// TwinCAT 3 PLC project Fraktal_Tests
// Title: Fraktal_Tests
// Company: fraktal-automation
// Author: fraktal-automation
// ProjectVersion: 0.1.0.10
// Description: Aggregate Fraktal Core + Modules + Press Demo TcUnit gate - excluded from deployed runtime (Core 5.7).
// ProgramVersion: 3.1.4026.24
// libraries:
//   Tc2_Standard, * (Beckhoff Automation GmbH)
//   Tc2_System, * (Beckhoff Automation GmbH)
//   Tc2_Utilities, * (Beckhoff Automation GmbH)
//   Tc3_Module, * (Beckhoff Automation GmbH)
//   Fraktal_Core, 0.3.0.0 (fraktal-automation)
//   Fraktal_Modules, 0.2.0.0 (fraktal-automation)
//   TcUnit, * (www.tcunit.org)
// project tree:
//   / PlcTask.TcTTO (not stored), FB_Access_Tests.TcPOU (not stored), FB_AlarmLog_Tests.TcPOU (not stored), FB_Base_Tests.TcPOU (not stored), FB_FaultRecovery_Tests.TcPOU, FB_ConfigurableCylinderCM_Tests.TcPOU (not stored), FB_ClampEM_Tests.TcPOU, FB_ClampStationUnit_Tests.TcPOU (not stored), FB_Connector_Tests.TcPOU (not stored), FB_CylinderCM_Tests.TcPOU, FB_Decision_Tests.TcPOU, FB_Hmi_Tests.TcPOU, FB_IoTopologyPublisher_Tests.TcPOU (not stored), FB_InputCM_Tests.TcPOU (not stored), FB_ManualCmd_Tests.TcPOU (not stored), FB_MultiRoot_Tests.TcPOU (not stored), FB_Oee_Tests.TcPOU (not stored), FB_PermIntlk_Tests.TcPOU (not stored), FB_PowerGroupCM_Tests.TcPOU (not stored), FB_TwoHandStartCM_Tests.TcPOU (not stored), FB_PressDemoUnit_Tests.TcPOU (not stored), FB_ProbeCM.TcPOU (not stored), FB_ProbeConnector.TcPOU (not stored), FB_ProbeEM.TcPOU (not stored), FB_ProbeUnit.TcPOU, FB_ProbeUnitManual.TcPOU (not stored), FB_Release_Tests.TcPOU (not stored), FB_PartTrace_Tests.TcPOU (not stored), FB_Shelve_Tests.TcPOU (not stored), FB_SystemInfrastructure_Tests.TcPOU (not stored), FB_TcpDev_Tests.TcPOU, FB_Timing_Tests.TcPOU (not stored), FB_Unit_Tests.TcPOU, PRG_TcUnitRunner.TcPOU
//   ../Fraktal_Press_Demo/01_PneumaticPress/Sequences/ FB_PressDemoLoadPosition.TcPOU (not stored), FB_PressDemoHome.TcPOU (not stored), FB_PressDemoChangeover.TcPOU (not stored), FB_PressDemoAuto.TcPOU
//   ../Fraktal_Press_Demo/01_PneumaticPress/Release/ FB_PressDemoRelease.TcPOU (not stored)
//   ../Fraktal_Press_Demo/01_PneumaticPress/ FB_PressDemoUnit.TcPOU
// (motion and I/O tree: see PLC project fraktal_press_demo)
// real-time tasks:
//   TASK PlcTask: cycle T#10ms, priority 20, ADS port 350
// variable links:

// ---- ../Fraktal_Press_Demo/01_PneumaticPress/Sequences/FB_PressDemoAuto.TcPOU
// AUTO mode chain (Core §6.2/§6.8 ST skeleton on FB_SequenceBase): the continuous
// production cycle — await a fresh two-hand start with part+air present, transfer
// the part in, press for the recipe dwell, return to load position, count the good
// part, and loop until Stop. A Stop requested at the between-cycles wait is honored
// there (M_StopNow) so no phantom cycle is charged. Every child motion goes through
// the §6.1 handshake (M_MayIssue); progression rides the shared _retVal.
FUNCTION_BLOCK FB_PressDemoAuto EXTENDS FB_SequenceBase
VAR
    _partReady, _airReady, _startReady : BOOL;
    _dwellTwoHandHeld : BOOL;          // N220 named wait: two-hand held through the dwell
    _traceAccepted, _recordAccepted, _partProcessed : BOOL;
    {attribute 'OPC.UA.DA' := '0'}
    _pressRam : REFERENCE TO FB_CylinderCM;
    {attribute 'OPC.UA.DA' := '0'}
    _door : REFERENCE TO FB_CylinderCM;
    {attribute 'OPC.UA.DA' := '0'}
    _partSlide : REFERENCE TO FB_CylinderCM;
    {attribute 'OPC.UA.DA' := '0'}
    _twoHand : REFERENCE TO FB_TwoHandStartCM;
    {attribute 'OPC.UA.DA' := '0'}
    _partPresentSensor : REFERENCE TO FB_DigitalInputCM;
    {attribute 'OPC.UA.DA' := '0'}
    _airPressureMonitor : REFERENCE TO FB_AirPressureMonitorCM;
    {attribute 'OPC.UA.DA' := '0'}
    _parCfg : REFERENCE TO ST_PneumaticPressParCfg;
    {attribute 'OPC.UA.DA' := '0'}
    _outCmd : REFERENCE TO ST_PneumaticPressOutCmd;
    {attribute 'OPC.UA.DA' := '0'}
    _startLatched : REFERENCE TO BOOL;
    {attribute 'OPC.UA.DA' := '0'}
    _loadPosition : FB_PressDemoLoadPosition;
    _loadPositionRunning : BOOL;
END_VAR

METHOD M_Reset
M_ResetBase(0);
_loadPositionRunning := FALSE;
_loadPosition.M_Reset(BaseStepNo := 0);
END_METHOD

METHOD M_Run
IF NOT _attached THEN
    RETURN;
END_IF
CASE _step OF
    0:  // initialize
        M_Step(StepNo := 0, StepName := 'project.step.pressAutoInitialize',
            Awaits := 0, AwaitingLabel := '', TimeClass := E_TimeClass.WORK, ExpectedTime := T#0S);
        _outCmd.CycleCompleted := FALSE;
        _outCmd.Homed := FALSE;
        _outCmd.ChangeoverCompleted := FALSE;
        _loadPositionRunning := FALSE;
        _retVal := E_StepResult.ADVANCE;
        M_Advance(OnAdvance := 100, OnJump1 := -1, OnJump2 := -1, OnJump3 := -1);
    100:  // await a fresh two-hand start (the §8.11.1 cycle-start marker)
        M_Step(StepNo := 100, StepName := 'project.step.pressAwaitTwoHand',
            Awaits := 0, AwaitingLabel := '', TimeClass := E_TimeClass.WAIT_OPERATOR, ExpectedTime := T#0S);
        _outCmd.CycleCompleted := FALSE;
        _partReady := M_Await(Idx := 1, Label := 'project.condition.partPresent',
            Ok := _partPresentSensor.OutImm.Value AND _partPresentSensor.OutImm.Quality);
        _airReady := M_Await(Idx := 2, Label := 'project.condition.airPressureOk',
            Ok := _airPressureMonitor.OutImm.PressureOk);
        IF _parCfg.RequireTwoHandStart THEN
            _startReady := M_Await(Idx := 3, Label := 'project.condition.twoHandStart', Ok := _startLatched);
        ELSE
            _startReady := TRUE;
        END_IF
        IF M_StopPending() THEN
            M_StopNow();                       // stop accepted BETWEEN cycles: no phantom cycle
        ELSIF _partReady AND _airReady AND _startReady THEN
            _traceAccepted := M_PartReceived();
            _retVal := E_StepResult.ADVANCE;
        END_IF
        M_Advance(OnAdvance := 110, OnJump1 := -1, OnJump2 := -1, OnJump3 := -1);
    110:  // ram up
        M_Step(StepNo := 110, StepName := 'project.step.pressRamUp',
            Awaits := _pressRam, AwaitingLabel := 'PressRam.RETRACT', TimeClass := E_TimeClass.WORK, ExpectedTime := T#0S);
        IF M_MayIssue(Steppable := TRUE) THEN
            _pressRam.Abort := FALSE; _pressRam.Command := E_CylinderCommand.RETRACT; _pressRam.Execute := TRUE;
        END_IF
        IF _pressRam.Done THEN _pressRam.Execute := FALSE; _retVal := E_StepResult.ADVANCE; END_IF
        M_Advance(OnAdvance := 130, OnJump1 := -1, OnJump2 := -1, OnJump3 := -1);
    130:  // door open
        M_Step(StepNo := 130, StepName := 'project.step.pressDoorOpen',
            Awaits := _door, AwaitingLabel := 'Door.RETRACT', TimeClass := E_TimeClass.WORK, ExpectedTime := T#0S);
        IF M_MayIssue(Steppable := TRUE) THEN
            _door.Abort := FALSE; _door.Command := E_CylinderCommand.RETRACT; _door.Execute := TRUE;
        END_IF
        IF _door.Done THEN _door.Execute := FALSE; _retVal := E_StepResult.ADVANCE; END_IF
        M_Advance(OnAdvance := 150, OnJump1 := -1, OnJump2 := -1, OnJump3 := -1);
    150:  // slide inside (value-adding sequence begins)
        M_Step(StepNo := 150, StepName := 'project.step.pressSlideInside',
            Awaits := _partSlide, AwaitingLabel := 'PartSlide.EXTEND', TimeClass := E_TimeClass.WORK, ExpectedTime := T#0S);
        IF M_MayIssue(Steppable := TRUE) THEN
            M_PartStarted();
            _partSlide.Abort := FALSE; _partSlide.Command := E_CylinderCommand.EXTEND; _partSlide.Execute := TRUE;
        END_IF
        IF _partSlide.Done THEN _partSlide.Execute := FALSE; _retVal := E_StepResult.ADVANCE; END_IF
        M_Advance(OnAdvance := 170, OnJump1 := -1, OnJump2 := -1, OnJump3 := -1);
    170:  // transfer settle
        M_Step(StepNo := 170, StepName := 'project.step.pressTransferSettle',
            Awaits := 0, AwaitingLabel := '', TimeClass := E_TimeClass.WORK, ExpectedTime := _parCfg.TransferSettleTime);
        _retVal := M_Delay(PT := _parCfg.TransferSettleTime);
        M_Advance(OnAdvance := 180, OnJump1 := -1, OnJump2 := -1, OnJump3 := -1);
    180:  // door close
        M_Step(StepNo := 180, StepName := 'project.step.pressDoorClose',
            Awaits := _door, AwaitingLabel := 'Door.EXTEND', TimeClass := E_TimeClass.WORK, ExpectedTime := T#0S);
        IF M_MayIssue(Steppable := TRUE) THEN
            _door.Abort := FALSE; _door.Command := E_CylinderCommand.EXTEND; _door.Execute := TRUE;
        END_IF
        IF _door.Done THEN _door.Execute := FALSE; _retVal := E_StepResult.ADVANCE; END_IF
        M_Advance(OnAdvance := 200, OnJump1 := -1, OnJump2 := -1, OnJump3 := -1);
    200:  // ram down
        M_Step(StepNo := 200, StepName := 'project.step.pressRamDown',
            Awaits := _pressRam, AwaitingLabel := 'PressRam.EXTEND', TimeClass := E_TimeClass.WORK, ExpectedTime := T#0S);
        IF M_MayIssue(Steppable := TRUE) THEN
            _pressRam.Abort := FALSE; _pressRam.Command := E_CylinderCommand.EXTEND; _pressRam.Execute := TRUE;
        END_IF
        IF _pressRam.Done THEN _pressRam.Execute := FALSE; _retVal := E_StepResult.ADVANCE; END_IF
        M_Advance(OnAdvance := 220, OnJump1 := -1, OnJump2 := -1, OnJump3 := -1);
    220:  // press dwell — two-hand must stay held; releasing it HOLDS the dwell
        M_Step(StepNo := 220, StepName := 'project.step.pressDwell',
            Awaits := 0, AwaitingLabel := '', TimeClass := E_TimeClass.WORK, ExpectedTime := _parCfg.PressSettleTime);
        // Releasing the button mid-dwell is the designed way to stop pressing, so it
        // is a named wait (§6.9(b)), not a fault: the ram's outputs come off, the
        // dwell timer freezes where it is because M_Delay is not called, and pressing
        // again restores the force and finishes the remaining dwell. Faulting here
        // charged an unrecoverable downtime event for normal operator behaviour.
        _dwellTwoHandHeld := M_Await(Idx := 1, Label := 'project.condition.twoHandHeldDuringPress',
            Ok := _twoHand.OutImm.SafeActive OR NOT _parCfg.RequireTwoHandStart);
        IF NOT _dwellTwoHandHeld THEN
            _pressRam.WithdrawOutputs();
        ELSE
            // The press force is the valve latched by the EXTEND that step 200 already
            // completed, so after a withdraw only this call re-energizes it — and the
            // ram re-checks its own extend permit before it does (§7.2).
            _pressRam.RestoreOutputs();
            _retVal := M_Delay(PT := _parCfg.PressSettleTime);
        END_IF
        M_Advance(OnAdvance := 230, OnJump1 := -1, OnJump2 := -1, OnJump3 := -1);
    230:  // record the applied dwell (§3.16.1 measured value)
        M_Step(StepNo := 230, StepName := 'project.step.pressRecordResult',
            Awaits := 0, AwaitingLabel := '', TimeClass := E_TimeClass.WORK, ExpectedTime := T#0S);
        _recordAccepted := M_PartRecord(RecordName := 'PressDwell',
            Value := DINT_TO_LREAL(TIME_TO_DINT(_parCfg.PressSettleTime)),
            Minimum := 0, Maximum := 30000,
            Target := DINT_TO_LREAL(TIME_TO_DINT(_parCfg.PressSettleTime)), EngUnit := 'ms');
        _loadPositionRunning := FALSE;
        _retVal := E_StepResult.ADVANCE;
        M_Advance(OnAdvance := 240, OnJump1 := -1, OnJump2 := -1, OnJump3 := -1);
    240:  // return to the shared load-safe position (composite step)
        IF NOT _loadPositionRunning THEN
            _loadPosition.M_Reset(BaseStepNo := 240);
            _loadPositionRunning := TRUE;
        END_IF
        _loadPosition.M_Run();
        IF _loadPosition.Done THEN
            _loadPositionRunning := FALSE;
            _retVal := E_StepResult.ADVANCE;
        END_IF
        M_Advance(OnAdvance := 999, OnJump1 := -1, OnJump2 := -1, OnJump3 := -1);
    999:  // cycle complete — write result, count by verdict, loop (§8.11.1 finish marker)
        M_Step(StepNo := 999, StepName := 'project.step.pressAutoComplete',
            Awaits := 0, AwaitingLabel := '', TimeClass := E_TimeClass.WORK, ExpectedTime := T#0S);
        _outCmd.CycleCompleted := TRUE;
        _partProcessed := M_PartProcessed(Verdict := E_Verdict.OK, Reason := E_Reason.NONE);
        IF NOT _partProcessed THEN
            M_CountGood();                     // §3.9: no carrier configured — count directly
        END_IF
        _startLatched := FALSE;
        IF M_EndOfCycle() THEN
            _retVal := E_StepResult.ADVANCE;   // stop NOT requested: loop to N100
        END_IF
        M_Advance(OnAdvance := 100, OnJump1 := -1, OnJump2 := -1, OnJump3 := -1);
ELSE
    M_Fault(Reason := E_Reason.STEP_STALLED, DescriptionKey := 'std.error.undefinedStep');
END_CASE
END_METHOD

METHOD Setup : BOOL
VAR_INPUT
    Host : I_SequenceHost;
END_VAR
VAR_IN_OUT
    PressRam : FB_CylinderCM;
    Door : FB_CylinderCM;
    PartSlide : FB_CylinderCM;
    TwoHand : FB_TwoHandStartCM;
    PartPresentSensor : FB_DigitalInputCM;
    AirPressureMonitor : FB_AirPressureMonitorCM;
    ParCfg : ST_PneumaticPressParCfg;
    OutCmd : ST_PneumaticPressOutCmd;
    StartLatched : BOOL;
END_VAR
_pressRam REF= PressRam;
_door REF= Door;
_partSlide REF= PartSlide;
_twoHand REF= TwoHand;
_partPresentSensor REF= PartPresentSensor;
_airPressureMonitor REF= AirPressureMonitor;
_parCfg REF= ParCfg;
_outCmd REF= OutCmd;
_startLatched REF= StartLatched;
Setup := M_Attach(Host := Host) AND __ISVALIDREF(_pressRam) AND __ISVALIDREF(_door)
    AND __ISVALIDREF(_partSlide) AND __ISVALIDREF(_twoHand)
    AND __ISVALIDREF(_partPresentSensor) AND __ISVALIDREF(_airPressureMonitor)
    AND __ISVALIDREF(_parCfg) AND __ISVALIDREF(_outCmd) AND __ISVALIDREF(_startLatched)
    AND _loadPosition.Setup(Host := Host, PressRam := PressRam, Door := Door, PartSlide := PartSlide);
END_METHOD

END_FUNCTION_BLOCK

// ---- ../Fraktal_Press_Demo/01_PneumaticPress/FB_PressDemoUnit.TcPOU
// Project-owned Unit: pneumatic press + access door + transfer slide + two-hand request.
// Cylinder interlocks prevent the two documented collisions in AUTO and MANUAL.
// Certified E-stop, two-hand evaluation and safe valve outputs remain external.
FUNCTION_BLOCK FB_PressDemoUnit EXTENDS FB_UnitBase
VAR_INPUT
    ParCfg : ST_PneumaticPressParCfg;
    ParCmd : ST_PneumaticPressParCmd;
END_VAR
VAR_OUTPUT
    PressRam      : FB_CylinderCM;
    Door          : FB_CylinderCM;
    PartSlide     : FB_CylinderCM;
    TwoHand       : FB_TwoHandStartCM;
    PneumaticPower: FB_PowerGroupCM;
    PartPresentSensor : FB_DigitalInputCM;
    AirPressureMonitor : FB_AirPressureMonitorCM;
    ReleaseConditions : FB_PressDemoRelease; // project-owned, browseable condition state
    OutCmd        : ST_PneumaticPressOutCmd;
    OutImm        : ST_PneumaticPressOutImm;
END_VAR
VAR
    {attribute 'OPC.UA.DA' := '0'}
    _recipe : I_RecipeProvider;
    _parCfgStaged : ST_PneumaticPressParCfg;
    _recipePrepared : BOOL;
    _startLatched : BOOL;
    _powerRequestPending : BOOL;
    _powerTargetOn : BOOL;
    {attribute 'OPC.UA.DA' := '0'}
    _homeSequence : FB_PressDemoHome;       // §6.8 ST chain on FB_SequenceBase owns HOME steps
    {attribute 'OPC.UA.DA' := '0'}
    _changeoverSequence : FB_PressDemoChangeover;
    {attribute 'OPC.UA.DA' := '0'}
    _autoSequence : FB_PressDemoAuto;
END_VAR

Cyclic();

METHOD Setup : BOOL
VAR_INPUT
    Name : STRING(80);
    PressHal : REFERENCE TO ST_CylinderHal;
    DoorHal : REFERENCE TO ST_CylinderHal;
    SlideHal : REFERENCE TO ST_CylinderHal;
    TwoHandHal : REFERENCE TO ST_TwoHandHal;
    PowerHal : REFERENCE TO ST_PowerGroupHal;
    PartPresentHal : REFERENCE TO ST_DigitalInputHal;
    AirPressureHal : REFERENCE TO ST_AirPressureHal;
    Recipe : I_RecipeProvider;
END_VAR
VAR
    InitialModel : ST_ModelId;
    Ok : BOOL;
END_VAR
_M_SetName(Name);
_M_SetPresentation(DisplayNameKey := 'project.module.pneumaticPress.name', DescriptionKey := 'project.module.pneumaticPress.description');
_recipe := Recipe;
Ok := PressRam.Setup(Name := CONCAT(Name, '.PressRam'), HalRef := PressHal, Recipe := 0);
Ok := Door.Setup(Name := CONCAT(Name, '.Door'), HalRef := DoorHal, Recipe := 0) AND Ok;
Ok := PartSlide.Setup(Name := CONCAT(Name, '.PartSlide'), HalRef := SlideHal, Recipe := 0) AND Ok;
Ok := TwoHand.Setup(Name := CONCAT(Name, '.TwoHand'), HalRef := TwoHandHal) AND Ok;
Ok := PneumaticPower.Setup(Name := CONCAT(Name, '.PneumaticPower'), HalRef := PowerHal) AND Ok;
Ok := PartPresentSensor.Setup(Name := CONCAT(Name, '.PartPresentSensor'),
    HalRef := PartPresentHal, DisplayNameKey := 'project.module.partPresentSensor.name',
    DescriptionKey := 'project.module.partPresentSensor.description') AND Ok;
Ok := AirPressureMonitor.Setup(Name := CONCAT(Name, '.AirPressureMonitor'),
    HalRef := AirPressureHal) AND Ok;
Ok := ReleaseConditions.Setup(UnitPath := Name) AND Ok;
Ok := _homeSequence.Setup(Host := THIS^, PressRam := PressRam, Door := Door,
    PartSlide := PartSlide, OutCmd := OutCmd) AND Ok;
Ok := _changeoverSequence.Setup(Host := THIS^, PressRam := PressRam, Door := Door,
    PartSlide := PartSlide, OutCmd := OutCmd, Model := Model) AND Ok;
Ok := _autoSequence.Setup(Host := THIS^, PressRam := PressRam, Door := Door,
    PartSlide := PartSlide, TwoHand := TwoHand, PartPresentSensor := PartPresentSensor,
    AirPressureMonitor := AirPressureMonitor, ParCfg := ParCfg, OutCmd := OutCmd,
    StartLatched := _startLatched) AND Ok;
PneumaticPower.ParCfg.Kind := E_PowerGroupKind.VALVE_ZONE;
PneumaticPower.ParCfg.RequiredForControl := TRUE;
PneumaticPower.ParCfg.FieldbusLossReaction := E_FieldbusLossReaction.CONTROL_OFF;
Ok := _M_Register(PressRam) AND Ok;
Ok := _M_Register(Door) AND Ok;
Ok := _M_Register(PartSlide) AND Ok;
Ok := _M_Register(TwoHand) AND Ok;
Ok := _M_Register(PneumaticPower) AND Ok;
Ok := _M_Register(PartPresentSensor) AND Ok;
Ok := _M_Register(AirPressureMonitor) AND Ok;
Setup := Ok AND PrepareRecipe(Model := InitialModel);
IF Setup THEN CommitRecipe(); END_IF
END_METHOD

METHOD PrepareRecipe : BOOL
VAR_INPUT
    Model : ST_ModelId;
END_VAR
IF _recipe = 0 THEN
    _parCfgStaged := ParCfg;
    _recipePrepared := TRUE;
ELSIF _recipe.Load(ModelCode := Model.ModelCode, RecipeKey := 'PneumaticPressUnit', pParCfg := ADR(_parCfgStaged), Size := SIZEOF(_parCfgStaged)) THEN
    IF (_parCfgStaged.PressSettleTime > T#30S) OR (_parCfgStaged.TransferSettleTime > T#5S) THEN
        _M_Fault(E_Reason.RECIPE_INVALID, 'project.error.pressRecipeInvalid');
        _recipePrepared := FALSE;
        PrepareRecipe := FALSE;
        RETURN;
    END_IF
    _recipePrepared := TRUE;
ELSE
    _M_Fault(E_Reason.RECIPE_INVALID, 'std.error.recipeSchemaInvalid');
    _recipePrepared := FALSE;
    PrepareRecipe := FALSE;
    RETURN;
END_IF
PrepareRecipe := SUPER^.PrepareRecipe(Model := Model);
IF NOT PrepareRecipe THEN _recipePrepared := FALSE; END_IF
END_METHOD

METHOD CommitRecipe
SUPER^.CommitRecipe();
IF _recipePrepared THEN
    ParCfg := _parCfgStaged;
    // §8.11 performance references follow the model: OEE Performance denominator
    // and the WORK-time degradation baseline are per-recipe engineering data.
    Oee.IdealCycleMs := ParCfg.IdealCycleMs;
    Profiler.M_SetBaselineWork(WorkMs := ParCfg.BaselineWorkMs);
END_IF
_recipePrepared := FALSE;
END_METHOD

METHOD AbortRecipe
SUPER^.AbortRecipe();
_recipePrepared := FALSE;
END_METHOD

// First operational scan: initialize application-owned mode-chain state.
METHOD PROTECTED OnInit : DINT
OnInit := SUPER^.OnInit();
_M_ResetModeSequences();
_M_ClearModeTransitionState();
END_METHOD

// Every accepted Unit Start gets a fresh mode chain, including a repeated
// HOME/CHANGEOVER run that does not pass through another mode change.
METHOD PROTECTED OnCommandStart : DINT
OnCommandStart := SUPER^.OnCommandStart();
_M_ResetModeSequences();
END_METHOD

// Mode-entry wiring only. Step behavior remains in the selected sequence POU.
METHOD PROTECTED OnModeChanged : DINT
VAR_INPUT
    NewMode : E_Mode;
    OldMode : E_Mode;
END_VAR
OnModeChanged := SUPER^.OnModeChanged(
    NewMode := NewMode, OldMode := OldMode);
_M_ResetModeSequences();
_M_ClearModeTransitionState();
END_METHOD

METHOD PROTECTED OnCyclic : DINT
OnCyclic := SUPER^.OnCyclic();
// Project release engineering is a separate visible component. It owns the
// functional collision permits and mode-entry conditions consumed below.
ReleaseConditions.M_Evaluate(PressRam := PressRam, Door := Door, PartSlide := PartSlide,
    TwoHand := TwoHand, PneumaticPower := PneumaticPower,
    AirPressure := AirPressureMonitor);

// Latch access-gated Unit requests, then observe one full Execute-low scan before
// starting another power-group command (PLCopen edge discipline).
IF ControlOffRequest THEN
    _powerTargetOn := FALSE;
    _powerRequestPending := TRUE;
ELSIF ControlOnRequest THEN
    _powerTargetOn := TRUE;
    _powerRequestPending := TRUE;
END_IF
IF PneumaticPower.Done OR PneumaticPower.Error OR PneumaticPower.Aborted THEN
    PneumaticPower.Execute := FALSE;
ELSIF _powerRequestPending AND NOT PneumaticPower.Execute
AND (PneumaticPower.State = E_ExecState.READY) THEN
    PneumaticPower.Abort := FALSE;
    IF _powerTargetOn THEN
        PneumaticPower.Command := E_PowerGroupCommand.POWER_ON;
    ELSE
        PneumaticPower.Command := E_PowerGroupCommand.POWER_OFF;
    END_IF
    PneumaticPower.Execute := TRUE;
    _powerRequestPending := FALSE;
END_IF

// A physical two-hand edge may start AUTO from READY, or release an already
// running Unit's wait step. It never bypasses domain readiness or access policy.
IF TwoHand.OutImm.StartPulse
AND PartPresentSensor.OutImm.Value AND PartPresentSensor.OutImm.Quality
AND AirPressureMonitor.OutImm.PressureOk THEN
    IF (State = E_ExecState.BUSY) AND (ModeActive = E_Mode.AUTO) THEN
        _startLatched := TRUE;
    ELSIF (ModeActive = E_Mode.AUTO) AND Start() THEN
        _startLatched := TRUE;
    END_IF
ELSIF TwoHand.OutImm.StartPulse THEN
    _startLatched := FALSE;
END_IF
IF PneumaticPower.Error AND (State = E_ExecState.BUSY) THEN
    _M_RollupFault();
END_IF
IF (State = E_ExecState.BUSY)
AND NOT AirPressureMonitor.OutImm.PressureOk THEN
    PressRam.WithdrawOutputs();
    Door.WithdrawOutputs();
    PartSlide.WithdrawOutputs();
    _M_Fault(E_Reason.PERMISSIVE_NOT_MET, 'project.error.pressAirPressureLost');
END_IF
OutImm.PressRetracted := PressRam.OutImm.Retracted;
OutImm.DoorOpen := Door.OutImm.Retracted;
OutImm.DoorClosed := Door.OutImm.Extended;
OutImm.SlideInside := PartSlide.OutImm.Extended;
OutImm.SlideOutside := PartSlide.OutImm.Retracted;
OutImm.TwoHandArmed := TwoHand.OutImm.Armed;
OutImm.TwoHandActive := TwoHand.OutImm.SafeActive;
OutImm.PartPresent := PartPresentSensor.OutImm.Value AND PartPresentSensor.OutImm.Quality;
OutImm.AirPressureOk := AirPressureMonitor.OutImm.PressureOk;
OutImm.ReadyForLoad := Door.OutImm.Retracted AND NOT Door.OutImm.Extended
    AND PartSlide.OutImm.Retracted AND NOT PartSlide.OutImm.Extended
    AND PressRam.OutImm.Retracted AND NOT PressRam.OutImm.Extended;
OutImm.ActiveSettleTime := ParCfg.PressSettleTime;
OutImm.Diagnostic := Status.Diagnostic;
END_METHOD

METHOD PROTECTED OnAbort : DINT
OnAbort := SUPER^.OnAbort();
_M_PartAborted();                    // §3.16.3: the part leaves without a valid result
_M_WithdrawSequenceOutputs();
_M_ResetModeSequences();
_M_ClearModeTransitionState();
_powerTargetOn := FALSE;
_powerRequestPending := TRUE;
END_METHOD

// Error-state Abort is a deliberate recovery action but does not clear ERROR.
METHOD PROTECTED OnAbortInError : DINT
OnAbortInError := SUPER^.OnAbortInError();
_M_WithdrawSequenceOutputs();
_M_ResetModeSequences();
_M_ClearModeTransitionState();
_powerTargetOn := FALSE;
_powerRequestPending := TRUE;
END_METHOD

// An operator reset is recovering this Unit: put the application back to the same
// safe wiring an error-state abort establishes, so the reset the operator presses at
// the panel needs no separate Stop/Abort first. The base then releases the run
// command and the children's commands, so the next HOME gets a genuine command edge.
// Unlike the abort paths this does NOT touch control power in either direction: it
// never requests Control On (§9.8 forbids self-resume), and it must not request
// Control Off either — powering down a healthy control circuit would make the
// operator re-enable it before HOME could run, i.e. reintroduce the multi-action
// recovery this reset exists to remove. Power stays where the operator put it.
METHOD PROTECTED OnOperatorReset : DINT
OnOperatorReset := SUPER^.OnOperatorReset();
_M_WithdrawSequenceOutputs();
_M_ResetModeSequences();
_M_ClearModeTransitionState();
END_METHOD

// One safe-stop wiring point shared by normal and error-state abort transitions.
METHOD PROTECTED _M_WithdrawSequenceOutputs
PressRam.WithdrawOutputs();
Door.WithdrawOutputs();
PartSlide.WithdrawOutputs();
PressRam.Execute := FALSE;
Door.Execute := FALSE;
PartSlide.Execute := FALSE;
END_METHOD

// Reset application-owned chain plumbing at lifecycle transitions. The chains'
// N000/N999 steps remain the only owners of process initialization/completion.
METHOD PROTECTED _M_ResetModeSequences
_homeSequence.M_Reset();
_changeoverSequence.M_Reset();
_autoSequence.M_Reset();
END_METHOD

// Clear state that must not survive init, mode entry, or either abort path.
// OnCommandStart deliberately does not call this: a physical start pulse may have
// been latched one scan before the inherited Execute edge is consumed.
METHOD PROTECTED _M_ClearModeTransitionState
Decision.Prompt := '';
DecisionAnswer := 0;
_startLatched := FALSE;
END_METHOD

// Application-only seam for ordinary hardwired Control On/Off buttons.
// It is a method (not OPC UA data), so HMI writes still use the access-gated
// ReqControlOn/ReqControlOff contract. The power CM rechecks safety and health.
METHOD RequestLocalControl : BOOL
VAR_INPUT
    ControlOn : BOOL;
END_VAR
_powerTargetOn := ControlOn;
_powerRequestPending := TRUE;
RequestLocalControl := TRUE;
END_METHOD

// §3.4.2 — the press paces every motion boundary through _M_StepGate, so
// SINGLE_STEP and HOLD_TO_RUN are supported (NON-SAFETY pacing; interlocks
// and the certified safety layer are unaffected).
METHOD PROTECTED _M_SupportsRunStyle : BOOL
VAR_INPUT
    Style : E_RunStyle;
END_VAR
_M_SupportsRunStyle := (Style = E_RunStyle.CONTINUOUS)
    OR (Style = E_RunStyle.SINGLE_STEP) OR (Style = E_RunStyle.HOLD_TO_RUN);
END_METHOD

METHOD PROTECTED _M_Supports : BOOL
VAR_INPUT
    Mode : E_Mode;
END_VAR
_M_Supports := (Mode = E_Mode.AUTO) OR (Mode = E_Mode.MANUAL)
    OR (Mode = E_Mode.HOME) OR (Mode = E_Mode.CHANGEOVER);
END_METHOD

// Thin mode router. Each supported sequence is a named method in the Unit tree.
METHOD PROTECTED _M_Dispatch
CASE ModeActive OF
    E_Mode.AUTO:
        _M_SequenceAuto();
    E_Mode.HOME:
        _M_SequenceHome();
    E_Mode.CHANGEOVER:
        _M_SequenceChangeover();
    E_Mode.MANUAL:
        _M_Fault(E_Reason.UNSUPPORTED_COMMAND, 'project.error.pressManualHasNoSequence');
ELSE
    _M_Fault(E_Reason.UNSUPPORTED_COMMAND, 'project.error.pressModeHasNoSequence');
END_CASE
END_METHOD

// Wiring-only HOME adapter. OnCommandStart owns the reset edge; the sequence POU
// owns every process step and terminal action.
METHOD PROTECTED _M_SequenceHome
_homeSequence.M_Run();
END_METHOD

// Wiring-only CHANGEOVER adapter. The §6.8 chain owns model validation, safe
// positioning, the operator decision, and completion logic.
METHOD PROTECTED _M_SequenceChangeover
_changeoverSequence.M_Run();
END_METHOD

// Wiring-only AUTO adapter. Every production command, wait, timer, decision,
// traceability action, and transition lives in the §6.8 chain.
METHOD PROTECTED _M_SequenceAuto
_autoSequence.M_Run();
END_METHOD

METHOD PROTECTED _M_RouteManual : BOOL
VAR_INPUT
    TargetPath : STRING(255);
    Value : DINT;
END_VAR
_M_RouteManual := FALSE;
IF TargetPath = PressRam.Name THEN
    _M_RouteManual := PressRam.ManualCommand(Value := Value);
ELSIF TargetPath = Door.Name THEN
    _M_RouteManual := Door.ManualCommand(Value := Value);
ELSIF TargetPath = PartSlide.Name THEN
    _M_RouteManual := PartSlide.ManualCommand(Value := Value);
ELSE
    _M_RouteManual := FALSE;
END_IF
END_METHOD

// §7.8 mode-entry release owned by this Unit. The base Start method consumes the
// same report the HMI displays, so this condition cannot become explanation-only.
METHOD PROTECTED _M_AppendInterlocks
VAR_IN_OUT
    Report : ST_ReleaseReport;
END_VAR
ReleaseConditions.M_AppendStart(Report := Report);
END_METHOD

METHOD PROTECTED _M_AppendManualInterlocks
VAR_INPUT
    TargetPath : STRING(255);
    Value : DINT;
END_VAR
VAR_IN_OUT
    Report : ST_ReleaseReport;
END_VAR
ReleaseConditions.M_AppendManual(TargetPath := TargetPath, Value := Value,
    PressRam := PressRam, Door := Door, PartSlide := PartSlide, Report := Report);
END_METHOD

METHOD PROTECTED _M_PublishStatus
SUPER^._M_PublishStatus();
OutImm.Diagnostic := Status.Diagnostic;
END_METHOD

// §3.10.2 — base walk (Unit facets + all child modules), then the project-owned
// fieldbus topology identity: static members of GVL_PressFieldbus.Topology are
// OPC.UA.DA=0 and reach the HMI only through this manifest.
METHOD M_AppendConfig : BOOL
VAR_INPUT
    Pager : REFERENCE TO FB_ConfigPager;
END_VAR
M_AppendConfig := SUPER^.M_AppendConfig(Pager := Pager);
F_AppendTopologyConfig(Topology := GVL_PressFieldbus.Topology, Pager := Pager);
END_METHOD

END_FUNCTION_BLOCK

// ---- FB_FaultRecovery_Tests.TcPOU
// Regression suite for the press hard-lock: an AUTO cycle reached N200 (ram down),
// the operator released the two-hand button mid-stroke — the designed way to stop a
// stroke — and NO panel action could recover the machine.
//
// Measured on the live PLC, the lock was two latches deep:
//   1. the lost permissive was classified as a FAULT, so the only exit was
//      Reset -> IDLE, and the fault's own condition ("two-hand held during a
//      stroke") could only be re-established by starting;
//   2. OperatorReset skipped an ACTIVE event and left both Execute inputs asserted,
//      and §6.1's Execute-drop reset — the sole exit from a latched terminal state —
//      needs them low. A Unit that is not BUSY never calls _M_Dispatch again, so the
//      frozen step holding `PressRam.Execute := TRUE` could never clear it, and the
//      next HOME re-issued an already-TRUE input: no rising edge, ram stuck in its
//      latched state, Unit re-adopting the fault through the §8.2 rollup.
//
// The ram is held mid-stroke deterministically by NOT calling its sim plant, so its
// position feedback never arrives (MoveTimeout is T#2S and a TON cannot advance
// inside one PLC scan, so it cannot expire here and turn the wait into a timeout).
FUNCTION_BLOCK FB_FaultRecovery_Tests EXTENDS TcUnit.FB_TestSuite
VAR
    Press : FB_PressDemoUnit;
    PressHal, DoorHal, SlideHal : ST_CylinderHal;
    TwoHandHal : ST_TwoHandHal;
    PowerHal : ST_PowerGroupHal;
    PartPresentHal : ST_DigitalInputHal;
    AirPressureHal : ST_AirPressureHal;
    PressSim, DoorSim, SlideSim : FB_CylinderSim;
    Recipe : FB_LocalRecipeProvider;
    Cfg : ST_PneumaticPressParCfg;
    Domain : ST_ControlDomainStatus;
    Release : ST_ReleaseReport;
    Wired : BOOL;
    i : INT;
END_VAR

IF NOT Wired THEN
    // A non-zero dwell keeps N220 open for the dwell-hold assertions; a TON never
    // advances inside a scan, so the dwell simply does not elapse during a test.
    Cfg.PressSettleTime := T#500MS;
    Cfg.TransferSettleTime := T#0S;
    Cfg.IdealCycleMs := 1000;
    Cfg.BaselineWorkMs := 900;
    Cfg.RequireTwoHandStart := TRUE;
    Recipe.Register(ModelCode := '', RecipeKey := 'PneumaticPressUnit', pData := ADR(Cfg), Size := SIZEOF(Cfg));
    PressHal.RetractedFb := TRUE; DoorHal.RetractedFb := TRUE; SlideHal.RetractedFb := TRUE;
    Press.Setup(Name := 'Test.Recovery', PressHal := PressHal, DoorHal := DoorHal,
        SlideHal := SlideHal, TwoHandHal := TwoHandHal, PowerHal := PowerHal,
        PartPresentHal := PartPresentHal, AirPressureHal := AirPressureHal, Recipe := Recipe);
    PressSim.Setup(HalRef := PressHal, TravelTime := T#0S);
    DoorSim.Setup(HalRef := DoorHal, TravelTime := T#0S);
    SlideSim.Setup(HalRef := SlideHal, TravelTime := T#0S);
    PowerHal.SafetyPermit := TRUE; PowerHal.FieldbusHealthy := TRUE; PowerHal.PowerFeedback := TRUE;
    TwoHandHal.FieldbusHealthy := TRUE;
    PartPresentHal.Quality := TRUE; PartPresentHal.Value := TRUE;
    AirPressureHal.Quality := TRUE;
    AirPressureHal.LowPressure := FALSE; AirPressureHal.OperatingPressure := TRUE;
    Domain.Present := TRUE; Domain.Id := 'TEST-RECOVERY'; Domain.ReadyForStart := TRUE;
    Domain.Safety.Present := TRUE; Domain.Safety.AllSafe := TRUE;
    Domain.ControlPower.Present := TRUE; Domain.ControlPower.ControlOn := TRUE;
    Press.ControlDomain := Domain;
    Press.SetMode(Mode := E_Mode.AUTO);
    Press();
    Wired := TRUE;
END_IF
Two_hand_release_mid_stroke_holds_the_ram();
Two_hand_release_in_the_dwell_holds_and_restores();
Latched_fault_recovers_with_one_operator_reset();
Reset_never_bypasses_a_live_condition();

// Drive the fixture from the load-safe position to N200 with the ram commanded
// EXTEND and still travelling. The ram's plant model is deliberately NOT ticked, so
// its extended feedback never arrives and the stroke stays in progress.
METHOD PROTECTED _M_RunToRamDown : BOOL
VAR
    scan : INT;
END_VAR
TwoHandHal.LeftPressed := FALSE; TwoHandHal.RightPressed := FALSE;
TwoHandHal.SafeActive := FALSE;
Press();                                     // clear any stale start pulse
TwoHandHal.LeftPressed := TRUE; TwoHandHal.RightPressed := TRUE;
TwoHandHal.SafeActive := TRUE;               // physical start edge (§3.4.2, non-safety)
FOR scan := 1 TO 40 DO
    DoorSim(); SlideSim(); Press();
END_FOR
_M_RunToRamDown := (Press.CurrentStep.StepNo = 200) AND Press.PressRam.Busy;
END_METHOD

// Leave the fixture where every test in this suite expects to find it: AUTO, stopped,
// no blocking event, ram/door/slide back at the load-safe position, two-hand released.
METHOD PROTECTED _M_ReturnToIdle
VAR
    scan : INT;
END_VAR
TwoHandHal.LeftPressed := FALSE; TwoHandHal.RightPressed := FALSE;
TwoHandHal.SafeActive := FALSE;
AirPressureHal.LowPressure := FALSE; AirPressureHal.OperatingPressure := TRUE;
Press.OperatorReset();
Press.Stop();
FOR scan := 1 TO 6 DO
    PressSim(); DoorSim(); SlideSim(); Press();
END_FOR
Press.SetMode(Mode := E_Mode.HOME);
Press();
Press.Start();
FOR scan := 1 TO 30 DO
    PressSim(); DoorSim(); SlideSim(); Press();
END_FOR
Press.Stop();
Press();
Press.SetMode(Mode := E_Mode.AUTO);
Press();
END_METHOD

// Defect B: releasing the button mid-stroke is expected operator behaviour, so it
// belongs in HELD (suspend, resume when restored), not in a fault whose only exit is
// Reset -> IDLE. Nothing is relaxed: the output is still withheld by the same permit.
METHOD Two_hand_release_mid_stroke_holds_the_ram
TEST('Two_hand_release_mid_stroke_holds_the_ram');
AssertTrue(Condition := _M_RunToRamDown(),
    Message := 'fixture reaches N200 with the ram travelling');
AssertTrue(Condition := PressHal.ExtendOut, Message := 'ram is driving down');

// The operator lets go, mid-stroke.
TwoHandHal.LeftPressed := FALSE; TwoHandHal.RightPressed := FALSE;
TwoHandHal.SafeActive := FALSE;
DoorSim(); SlideSim(); Press();
DoorSim(); SlideSim(); Press();

AssertFalse(Condition := PressHal.ExtendOut,
    Message := 'the permit still withholds the output — the interlock is untouched');
AssertTrue(Condition := Press.PressRam.Held, Message := 'ram is HELD (§6.1)');
AssertFalse(Condition := Press.PressRam.Error, Message := 'a released two-hand is not a ram fault');
AssertFalse(Condition := Press.Error, Message := 'and it is not a Unit fault either');
AssertFalse(Condition := Press.AlarmLog.Blocking,
    Message := 'no MANUAL_RESET event, so nothing blocks the restart (§8.3(b))');
AssertTrue(Condition := Press.Held, Message := 'the Unit reports the awaited hold (§8.2)');
AssertEquals_STRING(Expected := 'project.interlock.pressRequiresTwoHandHeld',
    Actual := Press.Status.Diagnostic.Description,
    Message := 'the operator sees WHICH condition is missing, not a composite key (§6.9)');
AssertEquals_STRING(Expected := 'Test.Recovery.PressRam',
    Actual := Press.Status.Diagnostic.SourcePath,
    Message := 'the held module names itself, not the Unit');

// Pressing again resumes the same stroke — no reset, no restart, no lost part.
TwoHandHal.LeftPressed := TRUE; TwoHandHal.RightPressed := TRUE;
TwoHandHal.SafeActive := TRUE;
DoorSim(); SlideSim(); Press();
AssertTrue(Condition := PressHal.ExtendOut, Message := 'resume re-energizes the ram');
AssertFalse(Condition := Press.PressRam.Held, Message := 'hold clears itself when the button returns');
FOR i := 1 TO 6 DO
    PressSim(); DoorSim(); SlideSim(); Press();      // let the stroke finish now
END_FOR
AssertEquals_INT(Expected := 220, Actual := Press.CurrentStep.StepNo,
    Message := 'the suspended stroke completes and the cycle carries on');
_M_ReturnToIdle();
TEST_FINISHED();
END_METHOD

// N220 holds the press force through the dwell. The force is the valve latched by the
// EXTEND that N200 already completed, so a withdraw needs an explicit restore — the
// case a hold at the CM alone does not cover.
METHOD Two_hand_release_in_the_dwell_holds_and_restores
TEST('Two_hand_release_in_the_dwell_holds_and_restores');
AssertTrue(Condition := _M_RunToRamDown(), Message := 'fixture reaches N200');
FOR i := 1 TO 6 DO
    PressSim(); DoorSim(); SlideSim(); Press();      // complete the stroke -> dwell
END_FOR
AssertEquals_INT(Expected := 220, Actual := Press.CurrentStep.StepNo, Message := 'dwelling at N220');
AssertTrue(Condition := PressHal.ExtendOut, Message := 'press force is applied during the dwell');

TwoHandHal.LeftPressed := FALSE; TwoHandHal.RightPressed := FALSE;
TwoHandHal.SafeActive := FALSE;
PressSim(); DoorSim(); SlideSim(); Press();
AssertFalse(Condition := PressHal.ExtendOut, Message := 'releasing the button stops pressing');
AssertFalse(Condition := Press.Error, Message := 'and does not fault the cycle');
AssertEquals_INT(Expected := 220, Actual := Press.CurrentStep.StepNo, Message := 'the dwell holds where it was');
AssertFalse(Condition := Press.CurrentStep.Conds[1].Ok,
    Message := 'the named dwell condition shows FALSE (§6.9(b))');

TwoHandHal.LeftPressed := TRUE; TwoHandHal.RightPressed := TRUE;
TwoHandHal.SafeActive := TRUE;
PressSim(); DoorSim(); SlideSim(); Press();
AssertTrue(Condition := PressHal.ExtendOut,
    Message := 'pressing again restores the press force (RestoreOutputs)');
_M_ReturnToIdle();
TEST_FINISHED();
END_METHOD

// Defect A + C, the actual hard-lock. Air loss mid-stroke is a genuine process fault
// (not an operator action), so it still faults — and that is exactly the state the
// press could not get out of. ONE reset has to make HOME runnable again.
METHOD Latched_fault_recovers_with_one_operator_reset
TEST('Latched_fault_recovers_with_one_operator_reset');
AssertTrue(Condition := _M_RunToRamDown(), Message := 'fixture reaches N200');

// Lose operating air while the ram is travelling: the Unit faults with the chain
// frozen at N200, which is where it had asserted PressRam.Execute.
AirPressureHal.OperatingPressure := FALSE;
AirPressureHal.LowPressure := TRUE;
DoorSim(); SlideSim(); Press();
DoorSim(); SlideSim(); Press();

AssertTrue(Condition := Press.Error, Message := 'air loss during motion is a real fault');
AssertTrue(Condition := Press.AlarmLog.Blocking, Message := 'and raises a blocking event (§8.3(b))');
AssertEquals_DINT(Expected := TO_DINT(E_AlarmState.ACTIVE),
    Actual := TO_DINT(Press.AlarmLog.Active[1].State),
    Message := 'the event is ACTIVE — it never reached WAIT_RESET');
// The two latches that made this unrecoverable:
AssertTrue(Condition := Press.Execute, Message := 'the run command is still asserted');
AssertTrue(Condition := Press.PressRam.Execute,
    Message := 'and so is the child command the frozen chain issued');

// Restore air: the CAUSE is gone, but the latched state is not, and Start stays shut.
AirPressureHal.OperatingPressure := TRUE;
AirPressureHal.LowPressure := FALSE;
DoorSim(); SlideSim(); Press();
Press.ReleaseReportStart(Report := Release);
AssertFalse(Condition := Release.Released,
    Message := 'a cleared cause does not by itself unlatch the Unit');

// ONE operator action.
AssertTrue(Condition := Press.OperatorReset(), Message := 'the reset is accepted');
AssertFalse(Condition := Press.AlarmLog.Blocking,
    Message := 'an ACTIVE MANUAL_RESET event closes on a deliberate reset (§8.3(b))');
AssertEquals_DINT(Expected := TO_DINT(E_AlarmState.CLOSED),
    Actual := TO_DINT(Press.AlarmLog.Active[1].State), Message := 'slot released');
AssertTrue(Condition := Press.AlarmLog.Ring[Press.AlarmLog.RingHead].Duration >= T#0S,
    Message := 'the closed event still carries a Duration (§8.3(a))');
AssertFalse(Condition := Press.Execute, Message := 'the stale run command is released');
AssertFalse(Condition := Press.PressRam.Execute, Message := 'the stranded child command is released');

DoorSim(); SlideSim(); Press();
DoorSim(); SlideSim(); Press();
AssertTrue(Condition := Press.State = E_ExecState.READY,
    Message := 'the Unit is READY after the inherited Execute-drop reset (§6.1)');
AssertTrue(Condition := Press.PressRam.State = E_ExecState.READY,
    Message := 'and so is the ram, so it can take a fresh command edge');

// Defect C: the recovery sequence is now reachable, under normal access authority.
AssertTrue(Condition := Press.SetMode(Mode := E_Mode.HOME), Message := 'HOME can be selected');
Press();
AssertTrue(Condition := Press.Start(), Message := 'HOME starts with no further operator action');
FOR i := 1 TO 30 DO
    PressSim(); DoorSim(); SlideSim(); Press();
END_FOR
AssertTrue(Condition := Press.OutCmd.Homed, Message := 'HOME reaches the load-safe position');
_M_ReturnToIdle();
TEST_FINISHED();
END_METHOD

// The reset closes a latched event even while its cause is unsatisfied, which is only
// safe because it clears the LATCH and never the condition. Proof: reset with the air
// still missing, then watch the release report keep Start shut on that live condition.
METHOD Reset_never_bypasses_a_live_condition
TEST('Reset_never_bypasses_a_live_condition');
AssertTrue(Condition := _M_RunToRamDown(), Message := 'fixture reaches N200');
AirPressureHal.OperatingPressure := FALSE;
AirPressureHal.LowPressure := TRUE;
DoorSim(); SlideSim(); Press();
DoorSim(); SlideSim(); Press();
AssertTrue(Condition := Press.AlarmLog.Blocking, Message := 'faulted with air missing');

AssertTrue(Condition := Press.OperatorReset(), Message := 'reset is accepted with the cause still live');
DoorSim(); SlideSim(); Press();
AssertFalse(Condition := Press.AlarmLog.Blocking, Message := 'the latch is cleared');
Press.ReleaseReportStart(Report := Release);
AssertFalse(Condition := Release.Released,
    Message := 'but Start is still refused — the reset cleared the latch, not the condition');
AssertFalse(Condition := Press.ReleaseConditions.ModeStartAirPressureOk,
    Message := 'and the live condition is still reported by name (§7.8)');
AssertFalse(Condition := PressHal.ExtendOut,
    Message := 'no output is restored by a reset');
_M_ReturnToIdle();
TEST_FINISHED();
END_METHOD

END_FUNCTION_BLOCK

// ---- FB_ClampEM_Tests.TcPOU
// Annex H §H.5 — the Composite (EM) tier suite.
//
// §5.7 coverage for this type. Rows T1/T4 and the T2/T6 *mechanisms* are proven
// once in the framework base suite (FB_Base_Tests) and are deliberately NOT
// re-tested here — "verification, like standardization, is paid once at the level
// that owns the behaviour". What this suite owes is the applicable rows re-proven
// with the TYPE's OWN reasons and source paths:
//   T2  first-out carries this type's reason + its own child path  (via T6 case)
//   T3  interlock withholds the output, with this type's path
//   T5  invalid ParCfg -> RECIPE_INVALID, never mis-runs
//   T6  cross-tier rollup: child first-out adopted verbatim  (composite row)
FUNCTION_BLOCK FB_ClampEM_Tests EXTENDS TcUnit.FB_TestSuite
VAR
    _em : FB_ClampEM;
    _hA, _hB : ST_CylinderHal;
    _simA : FB_CylinderSim;
    _pr : FB_LocalRecipeProvider;
    _bCyl : ST_CylinderParCfg;
    _bClamp : ST_ClampParCfg;
    _d : ST_Diagnostic;
    _w : BOOL;
    _i : INT;

    // T3 — a second EM whose CylA permissive is dropped before the command. It needs
    // its OWN cylinder recipe and plant: the shared record sets MoveTimeout := T#0S,
    // so the UNinterlocked partner used to time out in the same scan and the rollup
    // named CylA only because it happened to be first in registration order. With a
    // travel timeout the partner cannot expire, so this test now depends on the
    // interlock alone — and the sims let the suspended clamp finish after it returns.
    _emIntlk : FB_ClampEM;
    _hIA, _hIB : ST_CylinderHal;
    _simIntlkA, _simIntlkB : FB_CylinderSim;
    _prIntlk : FB_LocalRecipeProvider;
    _bCylTravel : ST_CylinderParCfg;

    // T5 — a third EM built on a recipe whose stored ClampEM schema is wrong.
    _emBad : FB_ClampEM;
    _hBA, _hBB : ST_CylinderHal;
    _prBad : FB_LocalRecipeProvider;
    _bClampBad : ST_ClampParCfg;
END_VAR

IF NOT _w THEN
    _bCyl.MoveTimeout := T#0S;               // CylB times out deterministically
    _bClamp.SettleTime := T#0S;
    _pr.Register(ModelCode := '', RecipeKey := 'CylinderCM', pData := ADR(_bCyl), Size := SIZEOF(_bCyl));
    _pr.Register(ModelCode := '', RecipeKey := 'ClampEM', pData := ADR(_bClamp), Size := SIZEOF(_bClamp));
    _em.Setup(Name := 'ClampStation', HalA := _hA, HalB := _hB, Recipe := _pr);
    _simA.Setup(HalRef := _hA, TravelTime := T#0S);
    _bCylTravel.MoveTimeout := T#5S;         // cannot expire inside a test scan
    _prIntlk.Register(ModelCode := '', RecipeKey := 'CylinderCM', pData := ADR(_bCylTravel), Size := SIZEOF(_bCylTravel));
    _prIntlk.Register(ModelCode := '', RecipeKey := 'ClampEM', pData := ADR(_bClamp), Size := SIZEOF(_bClamp));
    _emIntlk.Setup(Name := 'ClampIntlk', HalA := _hIA, HalB := _hIB, Recipe := _prIntlk);
    _simIntlkA.Setup(HalRef := _hIA, TravelTime := T#0S);
    _simIntlkB.Setup(HalRef := _hIB, TravelTime := T#0S);
    // Stored ClampEM record declares schema 2 while the type expects 1 (§3.8).
    _bClampBad.SchemaVersion := 2;
    _prBad.Register(ModelCode := '', RecipeKey := 'CylinderCM', pData := ADR(_bCyl), Size := SIZEOF(_bCyl));
    _prBad.Register(ModelCode := '', RecipeKey := 'ClampEM', pData := ADR(_bClampBad), Size := SIZEOF(_bClampBad));
    _w := TRUE;
END_IF
Clamp_rolls_up_CylB_first_out();
T3_interlock_withholds_child_output();
T5_recipe_schema_mismatch_faults();

METHOD Clamp_rolls_up_CylB_first_out
TEST('Clamp_rolls_up_CylB_first_out');
_em.Command := E_ClampCommand.CLAMP;
_em.Execute := TRUE;
FOR _i := 1 TO 6 DO
    _em();                                   // EM ticks children in OnCyclic
    _simA();                                 // plant completes CylA; CylB never arrives
END_FOR
AssertTrue(Condition := _em.Error, Message := 'EM faults on child error');
_d := _em.GetFaultSummary();
AssertEquals_DWORD(Expected := TO_DWORD(PL_ModuleReasons.CYL_NOT_EXTENDED),
                   Actual   := TO_DWORD(_d.ReasonCode),
                   Message  := 'EM adopts the child first-out verbatim (8.2)');
AssertEquals_STRING(Expected := 'ClampStation.CylB', Actual := _d.SourcePath,
                    Message := 'rollup names CylB, not the EM (H.5)');
TEST_FINISHED();
END_METHOD

// §5.7 T3 for the composite tier: a dropped permissive on a child must withhold
// the physical output and surface the interlock reason THROUGH the EM, naming the
// child that is actually blocked (not the EM) — the composite tier's own
// path/reason pairing, which the base-suite mechanism test cannot assert.
METHOD T3_interlock_withholds_child_output
TEST('T3_interlock_withholds_child_output');
_emIntlk.CylA.SimForceInterlock(Id := 1, Ok := FALSE);   // SIM-only hook (§5.7)
_emIntlk.Command := E_ClampCommand.CLAMP;
_emIntlk.Execute := TRUE;
FOR _i := 1 TO 4 DO
    _emIntlk();
END_FOR
AssertFalse(Condition := _hIA.ExtendOut,
    Message := 'interlocked child must not energize its output (§7)');
_d := _emIntlk.GetFaultSummary();
AssertEquals_DWORD(Expected := TO_DWORD(E_Reason.INTERLOCK_DROPPED),
    Actual := TO_DWORD(_d.ReasonCode),
    Message := 'EM surfaces the interlock reason (§7.2)');
AssertEquals_STRING(Expected := 'ClampIntlk.CylA', Actual := _d.SourcePath,
    Message := 'interlock names the blocked child, not the EM (§6.9)');
// §6.1 HELD rolls up like a fault does, but as information: the EM explains WHICH
// child waits on WHICH condition without entering ERROR or blocking a restart.
AssertTrue(Condition := _emIntlk.Held, Message := 'EM adopts the held child (§8.2)');
AssertFalse(Condition := _emIntlk.Error, Message := 'a held child does not fault the EM');
AssertFalse(Condition := _emIntlk.CylB.Error,
    Message := 'the partner keeps its command instead of being aborted');
// Restoring the condition resumes the join with no operator action.
_emIntlk.CylA.SimForceInterlock(Id := 1, Ok := TRUE);
FOR _i := 1 TO 6 DO
    _simIntlkA(); _simIntlkB(); _emIntlk();
END_FOR
AssertFalse(Condition := _emIntlk.Held, Message := 'hold clears itself when the child resumes');
AssertTrue(Condition := _emIntlk.OutCmd.Confirmed,
    Message := 'the suspended clamp completes after the interlock returns');
_emIntlk.Execute := FALSE;
_emIntlk();
TEST_FINISHED();
END_METHOD

// §5.7 T5 for the composite tier: a stored ClampEM ParCfg whose SchemaVersion is
// not the expected one must migrate-or-fault with RECIPE_INVALID and never
// mis-run with the wrong parameters (§3.8).
METHOD T5_recipe_schema_mismatch_faults
TEST('T5_recipe_schema_mismatch_faults');
// Setup resolves the recipe, so the fault is raised during construction.
_emBad.Setup(Name := 'ClampBad', HalA := _hBA, HalB := _hBB, Recipe := _prBad);
_emBad();                                    // map ErrorID
AssertTrue(Condition := _emBad.FaultActive,
    Message := 'migrate-or-fault on schema mismatch (§3.8)');
AssertEquals_DWORD(Expected := TO_DWORD(E_Reason.RECIPE_INVALID),
    Actual := _emBad.ErrorID,
    Message := 'RECIPE_INVALID on SchemaVersion mismatch (§3.8)');
// Never mis-runs: a command must not drive an output while the recipe is invalid.
_emBad.Command := E_ClampCommand.CLAMP;
_emBad.Execute := TRUE;
_emBad();
AssertFalse(Condition := _hBA.ExtendOut,
    Message := 'invalid recipe must not mis-run the actuator (§3.8)');
_emBad.Execute := FALSE;
_emBad();
TEST_FINISHED();
END_METHOD

END_FUNCTION_BLOCK

// ---- FB_CylinderCM_Tests.TcPOU
// Annex H suite for the cylinder TYPE: T2/T3/T5 with ITS reasons + functional
// completion against the sim plant model (T1/T4 inherited — not repeated, §5.7).
FUNCTION_BLOCK FB_CylinderCM_Tests EXTENDS TcUnit.FB_TestSuite
VAR
    _cm1, _cm2, _cm3, _cm4, _cm5, _cm6 : FB_CylinderCM;
    _h1, _h2, _h3, _h4, _h5, _h6 : ST_CylinderHal;
    _sim1 : FB_CylinderSim;
    _prOk, _prFast, _prBad : FB_LocalRecipeProvider;
    _bOk, _bFast, _bBad : ST_CylinderParCfg;
    _prModels : FB_LocalRecipeProvider;
    _modelA, _modelB, _loaded : ST_CylinderParCfg;
    _d : ST_Diagnostic;
    _release : ST_ReleaseReport;
    _io6 : ST_CylinderIoIdentity;
    _w : BOOL;
END_VAR

IF NOT _w THEN
    _bFast.MoveTimeout := T#0S;              // deterministic timeout in one scan
    _bBad.SchemaVersion := 2;                // stored schema != expected (=1)
    _prOk.Register(ModelCode := '', RecipeKey := 'CylinderCM', pData := ADR(_bOk), Size := SIZEOF(_bOk));
    _prFast.Register(ModelCode := '', RecipeKey := 'CylinderCM', pData := ADR(_bFast), Size := SIZEOF(_bFast));
    _prBad.Register(ModelCode := '', RecipeKey := 'CylinderCM', pData := ADR(_bBad), Size := SIZEOF(_bBad));
    _modelA.MoveTimeout := T#1S;
    _modelB.MoveTimeout := T#2S;
    _prModels.Register(ModelCode := 'A', RecipeKey := 'CylinderCM', pData := ADR(_modelA), Size := SIZEOF(_modelA));
    _prModels.Register(ModelCode := 'B', RecipeKey := 'CylinderCM', pData := ADR(_modelB), Size := SIZEOF(_modelB));
    _cm1.Setup(Name := 'Test.Cyl1', HalRef := _h1, Recipe := _prOk);
    _sim1.Setup(HalRef := _h1, TravelTime := T#0S);
    _cm2.Setup(Name := 'Test.Cyl2', HalRef := _h2, Recipe := _prFast);
    _cm3.Setup(Name := 'Test.Cyl3', HalRef := _h3, Recipe := _prOk);
    _cm5.Setup(Name := 'Test.Cyl5', HalRef := _h5, Recipe := _prOk);
    _cm6.Setup(Name := 'Test.Cyl6', HalRef := _h6, Recipe := _prFast);
    _io6.ExtendedSensor.Tag := '_101B202A';
    _io6.ExtendedSensor.Address := 'EL1809 Ch5';
    _io6.RetractedSensor.Tag := '_101B202B';
    _io6.RetractedSensor.Address := 'EL1809 Ch6';
    _io6.ExtendOutput.Tag := '_101K202A';
    _io6.RetractOutput.Tag := '_101K202B';
    _io6.ExtendedTimeoutKey := 'project.error.pressDownSensorTimeout';
    _io6.RetractedTimeoutKey := 'project.error.pressUpSensorTimeout';
    _io6.BothSensorsKey := 'project.error.pressPositionSensorsConflict';
    _cm6.ConfigureIoIdentity(Identity := _io6);
    _w := TRUE;
END_IF
Extend_completes_against_sim();
T2_first_out_reason_and_path();
T3_interlock_withholds_output();
T5_recipe_schema_mismatch_faults();
Recipe_lookup_uses_model_and_key();
Directional_interlock_covers_typed_command();
Timeout_identifies_sensor_tag();

METHOD Extend_completes_against_sim
TEST('Extend_completes_against_sim');
_cm1.Command := E_CylinderCommand.EXTEND;
_cm1.Execute := TRUE;
_cm1();                                      // edge -> step 10 drives ExtendOut
_cm1();                                      // step 20 awaiting fb
_sim1();                                     // plant: sensor made (travel T#0S)
_cm1();                                      // sees fb -> Done
AssertTrue(Condition := _cm1.Done, Message := 'handshake completes on feedback (6.1)');
AssertTrue(Condition := _cm1.Timing.Rows[1].Count = 1,
           Message := 'command timing row captured (8.11.4a)');
_cm1.Execute := FALSE;
_cm1();
TEST_FINISHED();
END_METHOD

METHOD Directional_interlock_covers_typed_command
TEST('Directional_interlock_covers_typed_command');
_cm5.SetDirectionalPermits(ExtendOk := FALSE, RetractOk := TRUE,
    ExtendDescriptionKey := 'project.interlock.testExtendBlocked',
    RetractDescriptionKey := 'project.interlock.testRetractAllowed');
_cm5.AppendDirectionalRelease(Value := TO_DINT(E_CylinderCommand.EXTEND), Report := _release);
AssertTrue(Condition := _release.Count = 1,
    Message := 'manual release query reports the selected blocked direction');
AssertEquals_STRING(Expected := 'project.interlock.testExtendBlocked',
    Actual := _release.Reasons[1].Description, Message := 'release query and dispatch share one key');
AssertEquals_STRING(Expected := 'Test.Cyl5', Actual := _release.Reasons[1].SourcePath,
    Message := 'directional release preserves the child module path');
_cm5.Command := E_CylinderCommand.EXTEND;
_cm5.Execute := TRUE;
_cm5();
AssertFalse(Condition := _h5.ExtendOut,
    Message := 'direction-specific collision interlock withholds output');
AssertEquals_DWORD(Expected := TO_DWORD(E_Reason.INTERLOCK_DROPPED),
    Actual := _cm5.ErrorID, Message := 'direction interlock uses common reason');
_d := _cm5.GetFaultSummary();
AssertEquals_STRING(Expected := 'project.interlock.testExtendBlocked',
    Actual := _d.Description, Message := 'selected direction publishes its key');
TEST_FINISHED();
END_METHOD

METHOD T2_first_out_reason_and_path
TEST('T2_first_out_reason_and_path');
_cm2.Command := E_CylinderCommand.EXTEND;
_cm2.Execute := TRUE;
_cm2();                                      // step 10
_cm2();                                      // step 20: MoveTimeout T#0S -> fault
AssertTrue(Condition := _cm2.Error, Message := 'Error after MoveTimeout');
AssertEquals_DWORD(Expected := TO_DWORD(PL_ModuleReasons.CYL_NOT_EXTENDED),
                   Actual   := _cm2.ErrorID,
                   Message  := 'first-out is the type band code 10101 (8.8)');
_d := _cm2.GetFaultSummary();
AssertEquals_STRING(Expected := 'Test.Cyl2', Actual := _d.SourcePath,
                    Message := 'reason names the source path (6.9)');
TEST_FINISHED();
END_METHOD

METHOD T3_interlock_withholds_output
TEST('T3_interlock_withholds_output');
_cm3.SimForceInterlock(Id := 1, Ok := FALSE);   // SIM-only hook (5.7)
_cm3.Command := E_CylinderCommand.EXTEND;
_cm3.Execute := TRUE;
_cm3();
AssertFalse(Condition := _h3.ExtendOut,
            Message := 'output must not energize while interlocked (7)');
AssertEquals_DWORD(Expected := TO_DWORD(E_Reason.INTERLOCK_DROPPED),
                   Actual   := _cm3.ErrorID,
                   Message  := 'interlock reason expected (7.2)');
_d := _cm3.GetFaultSummary();
AssertEquals_STRING(Expected := 'Test.Cyl3', Actual := _d.SourcePath,
                    Message := 'owner sets the source path (7.2)');
// 6.1 HELD — an interlock lost during a command suspends the command, it does not
// fail it: no ERROR to reset, no MANUAL_RESET alarm, and the reason is LOW.
AssertTrue(Condition := _cm3.Held, Message := 'interlocked command is HELD (6.1)');
AssertFalse(Condition := _cm3.Error, Message := 'a lost interlock is not a fault');
AssertTrue(Condition := _cm3.Busy, Message := 'held command stays BUSY so its owner keeps awaiting it');
AssertEquals_DINT(Expected := TO_DINT(E_Severity.LOW), Actual := TO_DINT(_d.Severity),
                  Message := 'a declared wait is LOW, not a downtime event (8.1/8.4)');
// ...and restoring the condition resumes it with no operator action at all.
_cm3.SimForceInterlock(Id := 1, Ok := TRUE);
_cm3();
AssertFalse(Condition := _cm3.Held, Message := 'hold clears itself when the condition returns');
AssertTrue(Condition := _h3.ExtendOut, Message := 'resume re-energizes the direction output');
AssertEquals_DWORD(Expected := 0, Actual := _cm3.ErrorID,
                   Message := 'the resumed command carries no lingering reason');
_cm3.Execute := FALSE;
_cm3();
TEST_FINISHED();
END_METHOD

METHOD T5_recipe_schema_mismatch_faults
TEST('T5_recipe_schema_mismatch_faults');
_cm4.Setup(Name := 'Test.Cyl4', HalRef := _h4, Recipe := _prBad);   // stored v2 vs expected v1
_cm4();                                      // map ErrorID
AssertTrue(Condition := _cm4.FaultActive, Message := 'migrate-or-fault (3.8)');
AssertEquals_DWORD(Expected := TO_DWORD(E_Reason.RECIPE_INVALID),
                   Actual   := _cm4.ErrorID,
                   Message  := 'RECIPE_INVALID on SchemaVersion mismatch (3.8)');
TEST_FINISHED();
END_METHOD

METHOD Recipe_lookup_uses_model_and_key
TEST('Recipe_lookup_uses_model_and_key');
AssertTrue(Condition := _prModels.Load(ModelCode := 'B', RecipeKey := 'CylinderCM',
    pParCfg := ADR(_loaded), Size := SIZEOF(_loaded)),
    Message := 'model-specific record found');
AssertTrue(Condition := _loaded.MoveTimeout = T#2S,
    Message := 'same recipe key resolves by ModelCode');
TEST_FINISHED();
END_METHOD

METHOD Timeout_identifies_sensor_tag
TEST('Timeout_identifies_sensor_tag');
_cm6.Command := E_CylinderCommand.EXTEND;
_cm6.Execute := TRUE;
_cm6();
_cm6();
_d := _cm6.GetFaultSummary();
AssertEquals_STRING(Expected := '_101B202A', Actual := _d.IoTag,
    Message := 'timeout carries exact schematic sensor tag');
AssertEquals_STRING(Expected := 'EL1809 Ch5', Actual := _d.IoAddress,
    Message := 'timeout carries terminal channel locator');
AssertEquals_STRING(Expected := 'project.error.pressDownSensorTimeout',
    Actual := _d.Description, Message := 'timeout uses project-localizable sensor message');
TEST_FINISHED();
END_METHOD

END_FUNCTION_BLOCK

// ---- FB_Decision_Tests.TcPOU
// Core §6.11: one active request, safe resolution, timeout/default and audit.
FUNCTION_BLOCK FB_Decision_Tests EXTENDS TcUnit.FB_TestSuite
VAR
    _operator : FB_ProbeUnit;
    _overlap  : FB_ProbeUnit;
    _timeout  : FB_ProbeUnit;
    _invalid  : FB_ProbeUnit;
    _operatorReq : ST_DecisionRequest;
    _overlapReq  : ST_DecisionRequest;
    _otherReq    : ST_DecisionRequest;
    _timeoutReq  : ST_DecisionRequest;
    _invalidReq  : ST_DecisionRequest;
    _report : ST_ReleaseReport;
    _wOperator, _wOverlap, _wTimeout, _wInvalid : BOOL;
    _ringHead : INT;
END_VAR

Operator_choice_is_validated_consumed_and_logged();
Repeated_request_is_idempotent_and_overlap_rejects();
Timeout_uses_the_validated_safe_default();
Invalid_timeout_default_faults_without_publication();

METHOD Operator_choice_is_validated_consumed_and_logged
VAR
    answer : INT;
END_VAR
TEST('Operator_choice_is_validated_consumed_and_logged');
IF NOT _wOperator THEN
    _operator.Setup(Name := 'Test.DecisionOperator');
    AssertTrue(Condition := _operator.Start(), Message := 'Unit starts');
    _operator();
    _operatorReq.Prompt := 'project.decision.operator';
    _operatorReq.Options[1] := 'project.option.retry';
    _operatorReq.Options[2] := 'project.option.continue';
    _operatorReq.Default := 1;
    _operatorReq.Timeout := T#5S;
    AssertTrue(Condition := _operator.M_TestAskDecision(Req := _operatorReq),
        Message := 'valid request is published');
    AssertTrue(Condition := _operator.SubmitDecision(Option := 2, Report := _report),
        Message := 'active published option is accepted through the authoritative entry');
    _operator();
    answer := _operator.M_TestTakeDecision();
    AssertEquals_INT(Expected := 2, Actual := answer,
        Message := 'answer is consumed exactly once');
    AssertEquals_STRING(Expected := '', Actual := _operator.Decision.Prompt,
        Message := 'consumption clears the complete public slot');
    AssertEquals_STRING(Expected := 'std.audit.decisionOperatorResolved option=2',
        Actual := _operator.AlarmLog.Ring[_operator.AlarmLog.RingHead].Description,
        Message := 'operator resolution is a domain audit event');
    _wOperator := TRUE;
END_IF
TEST_FINISHED();
END_METHOD

METHOD Repeated_request_is_idempotent_and_overlap_rejects
TEST('Repeated_request_is_idempotent_and_overlap_rejects');
IF NOT _wOverlap THEN
    _overlap.Setup(Name := 'Test.DecisionOverlap');
    AssertTrue(Condition := _overlap.Start(), Message := 'Unit starts');
    _overlap();
    _overlapReq.Prompt := 'project.decision.first';
    _overlapReq.Options[1] := 'project.option.ok';
    _overlapReq.Timeout := T#0S;
    _otherReq.Prompt := 'project.decision.second';
    _otherReq.Options[1] := 'project.option.cancel';
    _otherReq.Timeout := T#0S;
    AssertTrue(Condition := _overlap.M_TestAskDecision(Req := _overlapReq),
        Message := 'first request owns the slot');
    _ringHead := _overlap.AlarmLog.RingHead;
    AssertTrue(Condition := _overlap.M_TestAskDecision(Req := _overlapReq),
        Message := 'same request is idempotent');
    AssertEquals_INT(Expected := _ringHead, Actual := _overlap.AlarmLog.RingHead,
        Message := 'idempotent presentation does not duplicate request audit');
    AssertFalse(Condition := _overlap.M_TestAskDecision(Req := _otherReq),
        Message := 'different request cannot overwrite the active slot');
    AssertEquals_STRING(Expected := 'project.decision.first', Actual := _overlap.Decision.Prompt,
        Message := 'first producer retains ownership');
    AssertEquals_STRING(Expected := 'std.audit.decisionOverlapRejected',
        Actual := _overlap.AlarmLog.Ring[_overlap.AlarmLog.RingHead].Description,
        Message := 'overlap is rejected and logged');
    _ringHead := _overlap.AlarmLog.RingHead;
    AssertFalse(Condition := _overlap.M_TestAskDecision(Req := _otherReq),
        Message := 'repeated conflict remains rejected');
    AssertEquals_INT(Expected := _ringHead, Actual := _overlap.AlarmLog.RingHead,
        Message := 'one repeated producer cannot flood the bounded event ring');
    _overlap.M_TestClearDecision();
    _wOverlap := TRUE;
END_IF
TEST_FINISHED();
END_METHOD

METHOD Timeout_uses_the_validated_safe_default
VAR
    answer : INT;
END_VAR
TEST('Timeout_uses_the_validated_safe_default');
IF NOT _wTimeout THEN
    _timeout.Setup(Name := 'Test.DecisionTimeout');
    AssertTrue(Condition := _timeout.Start(), Message := 'Unit starts');
    _timeout();
    _timeoutReq.Prompt := 'project.decision.timeout';
    _timeoutReq.Options[1] := 'project.option.safeStop';
    _timeoutReq.Options[2] := 'project.option.continue';
    _timeoutReq.Default := 1;
    _timeoutReq.Timeout := T#1MS;
    AssertTrue(Condition := _timeout.M_TestAskDecision(Req := _timeoutReq),
        Message := 'timed request is published');
    _wTimeout := TRUE;
ELSE
    _timeout();
    IF _timeout.DecisionAnswer > 0 THEN
        answer := _timeout.M_TestTakeDecision();
        AssertEquals_INT(Expected := 1, Actual := answer,
            Message := 'timeout resolves to the validated safe default');
        AssertEquals_STRING(Expected := 'std.audit.decisionTimeoutResolved option=1',
            Actual := _timeout.AlarmLog.Ring[_timeout.AlarmLog.RingHead].Description,
            Message := 'timeout origin is explicit in the audit');
        TEST_FINISHED();
    END_IF
END_IF
END_METHOD

METHOD Invalid_timeout_default_faults_without_publication
TEST('Invalid_timeout_default_faults_without_publication');
IF NOT _wInvalid THEN
    _invalid.Setup(Name := 'Test.DecisionInvalid');
    AssertTrue(Condition := _invalid.Start(), Message := 'Unit starts');
    _invalid();
    _invalidReq.Prompt := 'project.decision.invalid';
    _invalidReq.Options[1] := 'project.option.safeStop';
    _invalidReq.Default := 2;
    _invalidReq.Timeout := T#1S;
    AssertFalse(Condition := _invalid.M_TestAskDecision(Req := _invalidReq),
        Message := 'missing default option is rejected');
    AssertTrue(Condition := _invalid.Error,
        Message := 'invalid application request faults instead of stalling silently');
    AssertEquals_STRING(Expected := '', Actual := _invalid.Decision.Prompt,
        Message := 'invalid request is never published');
    _wInvalid := TRUE;
END_IF
TEST_FINISHED();
END_METHOD

END_FUNCTION_BLOCK

// ---- FB_ProbeUnit.TcPOU
// minimal Unit for the base suite: 2-step looping chain, one wait-classed step
FUNCTION_BLOCK FB_ProbeUnit EXTENDS FB_UnitBase
VAR_INPUT
    SimA, SimB : BOOL;
    SimFault : BOOL;                    // deterministic fault injection for base-path tests
END_VAR
VAR_OUTPUT
    ModeChangedCount : UDINT;
    ModeExitCount : UDINT;
    ModeExitFirstCount : UDINT;
    LastNewMode : E_Mode;
    LastOldMode : E_Mode;
    LastRequestedMode : E_Mode;
END_VAR

Cyclic();

METHOD Setup : BOOL
VAR_INPUT
    Name : STRING(80);
END_VAR
_M_SetName(Name);
StallTime := T#0S;                       // test: stall pending fires immediately
Setup := TRUE;
END_METHOD

METHOD PROTECTED _M_Dispatch
CASE _step OF
    10:
        _M_SetStep(StepNo := 100, StepName := 'project.test.stepA', Awaits := 0,
            AwaitingLabel := '', Class := E_TimeClass.WORK, ExpectedTime := T#0S);
        IF SimFault THEN
            _M_Fault(E_Reason.TEST_FAULT, 'forced Unit fault');
        ELSIF SimA THEN
            _step := 20;
        END_IF
    20:
        _M_SetStep(StepNo := 200, StepName := 'project.test.stepB', Awaits := 0,
            AwaitingLabel := '', Class := E_TimeClass.WAIT_UPSTREAM, ExpectedTime := T#0S);
        IF SimB THEN
            _step := 30;
        END_IF
    30:
        IF _M_EndOfCycle() THEN
            _step := 10;
        END_IF
ELSE
    _M_Fault(E_Reason.STEP_STALLED, 'undefined step');
END_CASE
END_METHOD

// Test-probe seam for the protected §6.11 host service.
METHOD M_TestAskDecision : BOOL
VAR_INPUT
    Req : ST_DecisionRequest;
END_VAR
_M_AskDecision(Req := Req);
M_TestAskDecision := Decision.Prompt = Req.Prompt;
END_METHOD

METHOD M_TestClearDecision
M_SequenceClearDecision();
END_METHOD

METHOD M_TestTakeDecision : INT
M_TestTakeDecision := _M_TakeDecision();
END_METHOD

METHOD PROTECTED OnModeChanged : DINT
VAR_INPUT
    NewMode : E_Mode;
    OldMode : E_Mode;
END_VAR
OnModeChanged := SUPER^.OnModeChanged(
    NewMode := NewMode, OldMode := OldMode);
ModeChangedCount := ModeChangedCount + 1;
LastNewMode := NewMode;
LastOldMode := OldMode;
END_METHOD

METHOD PROTECTED OnModeExit : DINT
VAR_INPUT
    FirstCall : BOOL;
    RequestedMode : E_Mode;
END_VAR
// This probe wants the default immediate cancel, so the base call is intentional.
OnModeExit := SUPER^.OnModeExit(
    FirstCall := FirstCall, RequestedMode := RequestedMode);
ModeExitCount := ModeExitCount + 1;
IF FirstCall THEN
    ModeExitFirstCount := ModeExitFirstCount + 1;
END_IF
LastRequestedMode := RequestedMode;
END_METHOD

END_FUNCTION_BLOCK

// ---- FB_Hmi_Tests.TcPOU
// §3.10(a') under test: the data mirror IS the HMI contract — proven once.
FUNCTION_BLOCK FB_Hmi_Tests EXTENDS TcUnit.FB_TestSuite
VAR
    _p : FB_ProbeCM;
    _u : FB_ProbeUnit;
    _mailboxUnit : FB_ProbeUnit;
    _mailboxInit : BOOL;
    _policyUnit : FB_ProbeUnit;
    _policyInit : BOOL;
    _policyProvider : FB_LocalAccessProvider;
    _w : BOOL;
END_VAR

Status_mirror_carries_name_state_and_diag();
Unit_publishes_counters_and_history();
Nameplate_roundtrip();
Mailbox_commits_once_and_acknowledges();
Mailbox_policy_is_self_gated_and_power_ack_is_authoritative();

METHOD Status_mirror_carries_name_state_and_diag
TEST('Status_mirror_carries_name_state_and_diag');
IF NOT _w THEN
    _p.Setup('Test.Mirror');
    _u.Setup('Test.MirrorUnit');
    _w := TRUE;
END_IF
AssertEquals_STRING(Expected := 'Test.Mirror', Actual := _p.Status.Name,
                    Message := 'mirror carries the browse name (3.10a$')');
_p.Execute := TRUE;
_p.SimFault := TRUE;
_p();
AssertEquals_DINT(Expected := TO_DINT(E_ExecState.ERROR),
                  Actual   := TO_DINT(_p.Status.State),
                  Message  := 'mirror state follows ExecState');
AssertEquals_DWORD(Expected := TO_DWORD(E_Reason.TEST_FAULT),
                   Actual   := TO_DWORD(_p.Status.Diagnostic.ReasonCode),
                   Message  := 'live diagnostic published as DATA (6.9a)');
AssertTrue(Condition := _p.Status.FaultActive, Message := 'mirror fault flag');
_p.Execute := FALSE;
_p.SimFault := FALSE;
_p();
TEST_FINISHED();
END_METHOD

METHOD Unit_publishes_counters_and_history
TEST('Unit_publishes_counters_and_history');
_u.CountGood();
_u.CountGood();
_u.CountNok();
AssertEquals_UDINT(Expected := 2, Actual := _u.GoodCount, Message := 'good counter (8.11)');
AssertEquals_UDINT(Expected := 1, Actual := _u.NokCount,  Message := 'nok counter (8.11)');
// stall pending surfaces on the mirror while no fault is active (6.9/3.10a')
AssertTrue(Condition := _u.Start(), Message := 'start');
_u();
_u();                                        // StallTime T#0S -> pending
AssertEquals_DWORD(Expected := TO_DWORD(E_Reason.STEP_STALLED),
                   Actual   := TO_DWORD(_u.Status.Diagnostic.ReasonCode),
                   Message  := 'pending stall visible on the data mirror');
_u.Stop();
_u.SimA := TRUE;
_u.SimB := TRUE;
_u();
_u();
_u();
TEST_FINISHED();
END_METHOD

// §3.10.1: SetNameplate persists identity; published for the HMI facet card
METHOD Nameplate_roundtrip
VAR
    plate : ST_Nameplate;
END_VAR
TEST('Nameplate_roundtrip');
plate.ManufacturerName := 'ACME';
plate.SerialNumber := 'SN-1';
_p.SetNameplate(Plate := plate);
AssertEquals_STRING(Expected := 'ACME', Actual := _p.Nameplate.ManufacturerName, Message := 'manufacturer persists');
AssertEquals_STRING(Expected := 'SN-1', Actual := _p.Nameplate.SerialNumber, Message := 'serial persists');
TEST_FINISHED();
END_METHOD

// §3.10(a″): arguments are sampled only when Sequence changes; Ack is last.
METHOD Mailbox_commits_once_and_acknowledges
TEST('Mailbox_commits_once_and_acknowledges');
IF NOT _mailboxInit THEN
    _mailboxUnit.Setup('Test.MailboxUnit');
    _mailboxInit := TRUE;
ELSE
    _mailboxInit := _mailboxInit;
END_IF
_mailboxUnit.HmiRequest.Kind := E_HmiRequestKind.SET_MODE;
_mailboxUnit.HmiRequest.IntValue := TO_DINT(E_Mode.MANUAL);
_mailboxUnit.HmiRequest.Sequence := 1;
_mailboxUnit();
AssertEquals_UDINT(Expected := 1, Actual := _mailboxUnit.HmiResponse.AckSequence,
    Message := 'committed sequence acknowledged');
AssertTrue(Condition := _mailboxUnit.HmiResponse.Accepted,
    Message := 'existing gated SetMode path accepted');
AssertEquals_DINT(Expected := TO_DINT(E_Mode.MANUAL),
    Actual := TO_DINT(_mailboxUnit.ModeActivePublished),
    Message := 'property-only mode is published as OPC UA data');

// Change arguments without changing Sequence: the transaction shall not replay.
_mailboxUnit.HmiRequest.IntValue := TO_DINT(E_Mode.AUTO);
_mailboxUnit();
AssertEquals_DINT(Expected := TO_DINT(E_Mode.MANUAL),
    Actual := TO_DINT(_mailboxUnit.ModeActivePublished),
    Message := 'unchanged sequence is ignored');
TEST_FINISHED();
END_METHOD

METHOD Mailbox_policy_is_self_gated_and_power_ack_is_authoritative
TEST('Mailbox_policy_is_self_gated_and_power_ack_is_authoritative');
IF NOT _policyInit THEN
    _policyUnit.Setup('Test.PolicyMailboxUnit');
    _policyProvider.Register(User := 'admin1', Pin := '4711',
        Level := E_AccessLevel.ADMIN);
    _policyUnit();
    _policyUnit.Access.Setup(Provider := _policyProvider,
        pAlarmLog := ADR(_policyUnit.AlarmLog));
    _policyUnit.Access.ConfigureRequired(Gate := E_GatedAction.POWER_CONTROL,
        Level := E_AccessLevel.ADMIN);
    _policyInit := TRUE;
ELSE
    _policyInit := _policyInit;
END_IF

_policyUnit.HmiRequest.Kind := E_HmiRequestKind.CONTROL_ON;
_policyUnit.HmiRequest.Sequence := 1;
_policyUnit();
AssertFalse(Condition := _policyUnit.HmiResponse.Accepted,
    Message := 'control-power acknowledgement reflects PLC authorization');
AssertFalse(Condition := _policyUnit.ReqControlOn,
    Message := 'denied power request never latches');

_policyUnit.HmiRequest.Kind := E_HmiRequestKind.SET_ACCESS_LEVEL;
_policyUnit.HmiRequest.IntValue := TO_DINT(E_GatedAction.ACCESS_POLICY);
_policyUnit.HmiRequest.TextValue := '4';
_policyUnit.HmiRequest.Sequence := 2;
_policyUnit();
AssertFalse(Condition := _policyUnit.HmiResponse.Accepted,
    Message := 'anonymous session cannot raise ACCESS_POLICY above itself');
AssertEquals_DINT(Expected := TO_DINT(E_AccessLevel.NONE),
    Actual := TO_DINT(_policyUnit.Access.Policy.Required[TO_INT(E_GatedAction.ACCESS_POLICY)]),
    Message := 'self-lockout attempt leaves policy open');

_policyUnit.Access.RequestLogin(User := 'admin1', Secret := '4711');
_policyUnit();
_policyUnit.HmiRequest.Sequence := 3;
_policyUnit();
AssertTrue(Condition := _policyUnit.HmiResponse.Accepted,
    Message := 'authenticated admin may raise ACCESS_POLICY to ADMIN');
AssertEquals_DINT(Expected := TO_DINT(E_AccessLevel.ADMIN),
    Actual := TO_DINT(_policyUnit.Access.Policy.Required[TO_INT(E_GatedAction.ACCESS_POLICY)]),
    Message := 'ACCESS_POLICY threshold persisted');

_policyUnit.HmiRequest.IntValue := TO_DINT(E_GatedAction.DATA_WRITE);
_policyUnit.HmiRequest.TextValue := '2';
_policyUnit.Access.RequestLogout();
_policyUnit();
_policyUnit.HmiRequest.Sequence := 4;
_policyUnit();
AssertFalse(Condition := _policyUnit.HmiResponse.Accepted,
    Message := 'policy edits are self-gated after commissioning');
AssertEquals_DINT(Expected := TO_DINT(E_AccessLevel.NONE),
    Actual := TO_DINT(_policyUnit.Access.Policy.Required[TO_INT(E_GatedAction.DATA_WRITE)]),
    Message := 'denied edit leaves target threshold unchanged');
TEST_FINISHED();
END_METHOD

END_FUNCTION_BLOCK

// ---- FB_TcpDev_Tests.TcPOU
// Core §3.15.1a: CATEGORY CMs over the SIM channel — a generic vision CM is
// CONFIGURED (not subclassed) for an IV3-style dialect and parses judgement +
// payload; the reader CM parses code/NOREAD and verifies a match code; silence
// -> timeout fault 10402. No sockets, no vendor hardware.
FUNCTION_BLOCK FB_TcpDev_Tests EXTENDS TcUnit.FB_TestSuite
VAR
    _chan : FB_SimByteChannel;
    _vis  : FB_TcpVisionCM;
    _chanR: FB_SimByteChannel;
    _rdr  : FB_TcpCodeReaderCM;
    _chanT: FB_SimByteChannel;
    _visT : FB_TcpVisionCM;
    _chanIv3 : FB_SimByteChannel;
    _iv3 : FB_Iv3VisionCM;
    _chanMatrix : FB_SimByteChannel;
    _matrix : FB_Matrix220CM;
    _i    : INT;
    _w    : BOOL;
END_VAR

IF NOT _w THEN
    _chan.Script(Expect := 'T1$R', Reply := 'OK,123$R');
    _vis.Setup(Name := 'Test.Vision', Chan := _chan, DevHost := '10.0.0.5', DevPort := 9004);
    _vis.ParCfg.TriggerCmd := 'T1';                     // configured, not subclassed
    _chanR.Script(Expect := 'T$R', Reply := 'ABC-001$R');
    _rdr.Setup(Name := 'Test.Reader', Chan := _chanR, DevHost := '10.0.0.7', DevPort := 51236);
    _rdr.ParCmd.MatchCode := 'ABC-001';
    _visT.Setup(Name := 'Test.VisT', Chan := _chanT, DevHost := '10.0.0.6', DevPort := 9004);
    _visT.ParCfg.RespTimeout := T#40MS;
    _iv3.Setup(Name := 'Test.IV3', Chan := _chanIv3, DevHost := '10.0.0.8', DevPort := 9004);
    _matrix.Setup(Name := 'Test.Matrix220', Chan := _chanMatrix, DevHost := '10.0.0.9', DevPort := 51236);
    _w := TRUE;
END_IF
Vision_configured_parses();
Reader_code_and_match();
Timeout_faults_10402();
Model_presets_apply_configuration();

METHOD Vision_configured_parses
TEST('Vision_configured_parses');
_vis();
_vis.SendRequest(Text := _vis.ParCfg.TriggerCmd);
_vis();
AssertTrue(Condition := _vis.OutCmd.JudgeOk, Message := 'OK judgement parsed by the CATEGORY CM');
AssertEquals_STRING(Expected := '123', Actual := _vis.OutCmd.ResultData, Message := 'payload after prefix+separator');
TEST_FINISHED();
END_METHOD

METHOD Reader_code_and_match
TEST('Reader_code_and_match');
_rdr();
_rdr.SendRequest(Text := _rdr.ParCfg.TriggerCmd);
_rdr();
AssertEquals_STRING(Expected := 'ABC-001', Actual := _rdr.OutCmd.Code, Message := 'decoded symbol published');
AssertFalse(Condition := _rdr.OutCmd.NoRead, Message := 'not a no-read');
AssertTrue(Condition := _rdr.OutCmd.MatchOk, Message := 'configured match code verified');
TEST_FINISHED();
END_METHOD

METHOD Timeout_faults_10402
TEST('Timeout_faults_10402');
_visT();
IF NOT _visT.Error AND _i = 0 THEN
    _chanT.SwallowNext := TRUE;
    _visT.SendRequest(Text := _visT.ParCfg.TriggerCmd);
    _i := 1;
END_IF
_visT();
IF _visT.Error THEN
    AssertEquals_DWORD(Expected := TO_DWORD(PL_TcpDevReasons.DEV_RESP_TIMEOUT),
                       Actual := _visT.ErrorID, Message := 'silence -> 10402');
    TEST_FINISHED();
END_IF
END_METHOD

// §5.7: every released reusable type earns an automated check. These two types
// are configuration-only model presets, so their owned behavior is the preset
// values plus propagation of the endpoint through SUPER^.Setup.
METHOD Model_presets_apply_configuration
TEST('Model_presets_apply_configuration');
AssertEquals_STRING(Expected := 'T1', Actual := _iv3.ParCfg.TriggerCmd,
    Message := 'IV3 preset owns its verified trigger string');
AssertEquals_STRING(Expected := 'OK', Actual := _iv3.ParCfg.OkPrefix,
    Message := 'IV3 preset owns its OK prefix');
AssertEquals_STRING(Expected := '10.0.0.8', Actual := _iv3.ParCfg.Host,
    Message := 'IV3 preset still calls the category Setup');
AssertEquals_STRING(Expected := 'T', Actual := _matrix.ParCfg.TriggerCmd,
    Message := 'Matrix 220 preset owns its trigger string');
AssertEquals_STRING(Expected := 'NOREAD', Actual := _matrix.ParCfg.NoReadText,
    Message := 'Matrix 220 preset owns its no-read token');
AssertEquals_STRING(Expected := '10.0.0.9', Actual := _matrix.ParCfg.Host,
    Message := 'Matrix 220 preset still calls the category Setup');
TEST_FINISHED();
END_METHOD

END_FUNCTION_BLOCK

// ---- FB_Unit_Tests.TcPOU
// FB_UnitBase suite: mode rejection, run-as-command, stall key, wait-class
// derived Starved, cycle publication, mode change = immediate software abort by default.
FUNCTION_BLOCK FB_Unit_Tests EXTENDS TcUnit.FB_TestSuite
VAR
    _u : FB_ProbeUnit;
    _w : BOOL;
    _pager : FB_ConfigPager;
    _page : ST_ConfigPage;
END_VAR

Unit_run_stall_classes_and_cycle();
Unit_mode_change_is_estop_by_default();
Unit_config_capability_is_typed_and_fail_closed();

METHOD Unit_run_stall_classes_and_cycle
TEST('Unit_run_stall_classes_and_cycle');
IF NOT _w THEN
    _u.Setup('Test.Unit');
    _w := TRUE;
END_IF
AssertFalse(Condition := _u.SetMode(Mode := E_Mode.CALIBRATION),
            Message := 'unsupported mode rejected gracefully (3.4/3.7)');
AssertTrue(Condition := _u.Start(), Message := 'Start issues the run command (6 intro)');
_u();                                         // edge -> BUSY, step 100 set
_u();                                         // stall guard (T#0S) fires -> pending
AssertTrue(Condition := _u.Busy, Message := 'running');
AssertEquals_DWORD(Expected := TO_DWORD(E_Reason.STEP_STALLED),
                   Actual   := TO_DWORD(_u.Pending.ReasonCode),
                   Message  := 'stall is a PENDING reason, not a fault (6.9)');
AssertEquals_STRING(Expected := 'std.diagnostic.stepStalled',
                    Actual   := _u.Pending.Description,
                    Message  := 'stall publishes a stable key; CurrentStep carries context');
AssertFalse(Condition := _u.Error, Message := 'no fault from a stall');
_u.SimA := TRUE;
_u();                                         // -> step 200 (WAIT_UPSTREAM)
_u();
AssertTrue(Condition := _u.Starved,
           Message := 'Starved derived from the step wait class (8.11.4f/8.11.3)');
_u.Stop();
_u.SimB := TRUE;
_u();                                         // -> step 30
_u();                                         // EndOfCycle: publish + complete + release
_u();                                         // reset -> READY
AssertFalse(Condition := _u.Busy, Message := 'stopped after cycle (3.3)');
AssertEquals_INT(Expected := 2, Actual := _u.Profiler.LastCycle.NSteps,
                 Message := 'cycle profile published with both steps (8.11.4b)');
TEST_FINISHED();
END_METHOD

METHOD Unit_config_capability_is_typed_and_fail_closed
VAR
    i : INT;
    found : BOOL;
END_VAR
TEST('Unit_config_capability_is_typed_and_fail_closed');
_pager.M_Setup(Target := ADR(_page), PageIndex := 0, Revision := 1);
_u.M_AppendConfig(Pager := _pager);
_pager.M_Finish();
FOR i := 1 TO _page.EntryCount DO
    IF _page.Entries[i].WriteKey = 'unit.modePolicy.3.shield' THEN
        found := TRUE;
        AssertTrue(Condition := _page.Entries[i].Writable,
            Message := 'mode policy is an explicit write capability');
        AssertEquals_UDINT(Expected := 1, Actual := _page.Entries[i].WriteRevision,
            Message := 'write capability has a non-zero schema revision');
        AssertTrue(Condition := _page.Entries[i].RequiresReady,
            Message := 'capability publishes its READY-state constraint');
    END_IF
END_FOR
AssertTrue(Condition := found, Message := 'stable mode-policy key is manifest-served');
AssertTrue(Condition := _u.WriteConfig(TargetPath := 'Test.Unit',
    WriteKey := 'unit.modePolicy.3.shield', Revision := 1, TextValue := '0'),
    Message := 'registered exact enum value is accepted while READY');
AssertEquals_DINT(Expected := TO_DINT(E_ModeSwitchShield.INTERRUPTIBLE),
    Actual := TO_DINT(_u.ModePolicy[3].Shield), Message := 'typed handler applied value');
AssertFalse(Condition := _u.WriteConfig(TargetPath := 'Test.Unit',
    WriteKey := 'unit.modePolicy.3.shield', Revision := 2, TextValue := '1'),
    Message := 'stale capability revision is rejected');
AssertFalse(Condition := _u.WriteConfig(TargetPath := 'Test.Unit',
    WriteKey := 'unit.modePolicy.3.shield', Revision := 1, TextValue := '9'),
    Message := 'out-of-domain value is rejected');
AssertFalse(Condition := _u.WriteConfig(TargetPath := 'Other.Unit',
    WriteKey := 'unit.modePolicy.3.shield', Revision := 1, TextValue := '1'),
    Message := 'foreign owner path is rejected');
TEST_FINISHED();
END_METHOD

METHOD Unit_mode_change_is_estop_by_default
TEST('Unit_mode_change_is_estop_by_default');
_u.SimA := FALSE;
_u.SimB := FALSE;
AssertTrue(Condition := _u.Start(), Message := 're-start');
_u();
AssertTrue(Condition := _u.Busy, Message := 'running again');
AssertTrue(Condition := _u.SetMode(Mode := E_Mode.MANUAL), Message := 'mode request accepted (pending)');
_u();                                         // OnModeExit=0 -> OnAbort (non-safety software abort, 3.14.4)
_u();                                         // release run command, reset
_u();                                         // commit mode
AssertFalse(Condition := _u.Busy, Message := 'chain cancelled by the mode change');
AssertEquals_UDINT(Expected := 1, Actual := _u.ModeExitCount,
    Message := 'OnModeExit runs once for this immediate transition');
AssertEquals_UDINT(Expected := 1, Actual := _u.ModeExitFirstCount,
    Message := 'OnModeExit receives FirstCall exactly once');
AssertEquals_DINT(Expected := TO_DINT(E_Mode.MANUAL),
    Actual := TO_DINT(_u.LastRequestedMode),
    Message := 'OnModeExit receives the pending target mode');
AssertEquals_UDINT(Expected := 1, Actual := _u.ModeChangedCount,
    Message := 'OnModeChanged runs once after commit');
AssertEquals_DINT(Expected := TO_DINT(E_Mode.AUTO),
    Actual := TO_DINT(_u.LastOldMode),
    Message := 'OnModeChanged receives the mode being left');
AssertEquals_DINT(Expected := TO_DINT(E_Mode.MANUAL),
    Actual := TO_DINT(_u.LastNewMode),
    Message := 'OnModeChanged receives the committed mode');
AssertEquals_DINT(Expected := TO_DINT(E_Mode.MANUAL),
                  Actual   := TO_DINT(_u.ModeActive),
                  Message  := 'mode committed after leaving BUSY (3.14.4)');
TEST_FINISHED();
END_METHOD

END_FUNCTION_BLOCK

// ---- PRG_TcUnitRunner.TcPOU
// Core §5.7 / TC3 §5.7 — one open-ended gate: every suite joins unchanged (§6.8, H.6)
PROGRAM PRG_TcUnitRunner
VAR
    BaseTests      : FB_Base_Tests;
    PermTests      : FB_PermIntlk_Tests;
    PowerGroupTests: FB_PowerGroupCM_Tests;
    TwoHandTests   : FB_TwoHandStartCM_Tests;
    PressDemoTests : FB_PressDemoUnit_Tests;
    TimingTests    : FB_Timing_Tests;
    UnitTests      : FB_Unit_Tests;
    ConnectorTests : FB_Connector_Tests;
    CylinderTests  : FB_CylinderCM_Tests;
    DecisionTests  : FB_Decision_Tests;
    ConfigurableCylinderTests : FB_ConfigurableCylinderCM_Tests;
    ClampTests     : FB_ClampEM_Tests;
    ClampStationTests : FB_ClampStationUnit_Tests;
    HmiTests       : FB_Hmi_Tests;
    IoTopologyTests: FB_IoTopologyPublisher_Tests;
    InputModuleTests: FB_InputCM_Tests;
    AccessTests    : FB_Access_Tests;
    AlarmLogTests  : FB_AlarmLog_Tests;
    ManualCmdTests : FB_ManualCmd_Tests;
    MultiRootTests : FB_MultiRoot_Tests;
    OeeTests       : FB_Oee_Tests;
    ReleaseTests   : FB_Release_Tests;
    ShelveTests    : FB_Shelve_Tests;
    TcpDeviceTests : FB_TcpDev_Tests;
    PartTraceTests : FB_PartTrace_Tests;
    FaultRecoveryTests : FB_FaultRecovery_Tests;
    SystemInfrastructureTests : FB_SystemInfrastructure_Tests;
END_VAR

TcUnit.RUN();

END_PROGRAM
